	sCSVLine		: T_MaxString := '';(* Single CSV text line (row, record), we are using string as record buffer (your are able to see created fields) *)
	sCSVField		: T_MaxString := '';(* Single CSV field value (column, record field) *)
	//sCSVField		: UDINT;

	nRow	 		: UDINT 	:= 0;(* Row number (record) *)
	nColumn			: UDINT 	:= 0;(* Column number (record field) *)
	hFile			: UINT		:= 0;(* File handle of the source file *)
	step			: DWORD 	:= 0;
	fbFileOpen		: FB_FileOpen;(* Opens file *)
	fbFileClose		: FB_FileClose;(* Closes file *)
	fbFilePuts		: FB_FilePuts;(* Writes one record (line) *)
	fbFileWrite     : FB_FileWrite;
	fbWriter		: FB_CSVMemBufferWriter;(* Helper function block used to create CSV data bytes (single record line) *)
    StringModelWrite		: StringModel_256000_EX;
	fbFileRename			: FB_FileRename;//修改文件名称
	fbFileDelete			: FB_FileDelete;//删除文件
	writeTON				: TON;//延时写入

	(* :=[ (* Source PLC database *)
	'0_0', '0_1', '0_2', '0_3', '0_4', '0_5',
	'1_0', '1_1', '1_2', '1_3', '1_4', '1_5',
	'2_0', '2_1', '2_2', '2_3', '2_4', '2_5',
	'3_0', '3_1', '3_2', '3_3', '3_4', '3_5',
	'4_0', '4_1', '4_2', '4_3', '4_4', '4_5',
	'5_0', '5_1', '5_2', '5_3', '5_4', '5_5'];*)

END_VAR

DEFAULT_CSV_FIELD_SEP:= 16#2C;  //配置CSV文件的分割符，16#2C表明各个参数之间是用逗号分隔的。
CASE step OF
	0:(* Wait for rising edge at bWrite variable *)
		IF bWrite THEN
			bWrite 	:= FALSE;
			bBusy 	:= TRUE;
			error	:= FALSE;
			bError	:= FALSE;
			nErrId	:= 0;
			hFile	:= 0;
			nRow	:= 0;
			nColumn	:= 0;
			step 	:= 1;
		END_IF
	1:
		StringModelWrite.init();
		fbFileDelete(bExecute:= FALSE);
		fbFileRename(bExecute:= FALSE);
		step:=2;
	2:
		fbFileDelete(
			sNetId:= , 
			sPathName:= sFileNameOld, 
			ePath:= PATH_GENERIC, 
			bExecute:= TRUE, 
			tTimeout:= DEFAULT_ADS_TIMEOUT, 
			bBusy=> , 
			bError=> , 
			nErrId=> );
		step:=3;
	3:
		fbFileDelete(bExecute:= FALSE);
		IF NOT fbFileDelete.bBusy THEN
			step:=4;
		END_IF
	4:
		fbFileRename(
			sNetId:= , 
			sOldName:= sFileName, 
			sNewName:= sFileNameOld, 
			ePath:= PATH_GENERIC, 
			bExecute:= TRUE, 
			tTimeout:= DEFAULT_ADS_TIMEOUT, 
			bBusy=> , 
			bError=> , 
			nErrId=> );
		step:=5;
	5:
		fbFileRename(bExecute:= FALSE);
		IF NOT fbFileRename.bBusy THEN
			step:=10;
		END_IF

	10:(* Open source file *)
		fbFileOpen(  bExecute := FALSE  );
		fbFileOpen( sNetId := sNetId, sPathName := sFileName, nMode := FOPEN_MODEWRITE OR FOPEN_MODETEXT,(* Open file in TEXT mode! *)
					ePath := PATH_GENERIC, bExecute := TRUE );
		step := 20;

	20:(* Wait until open not busy *)
		//StringModelWrite.init();
		fbFileOpen( bExecute := FALSE, bError => bError, nErrID => nErrID, hFile => hFile );
		IF NOT fbFileOpen.bBusy THEN
			IF NOT fbFileOpen.bError THEN
				step := 30;
			ELSE(* Error: file not found? *)
				step := 1000;
			END_IF
		END_IF
	
	30:(* Convert one PLC record to CSV format *)
		FOR nRow:=0 TO csv_rows BY 1 DO
				sCSVLine := '';
				fbWriter.eCmd := eEnumCmd_First;(* Write first field value *)
			FOR nColumn := 0 TO csv_columns BY 1 DO
				sCSVField := STRING_TO_CSVFIELD( database[ nRow, nColumn ], FALSE );(* TODO: Get field value from your application *)
				(* Add new field to the record buffer *)
				fbWriter( 	pBuffer := ADR( sCSVLine ), cbBuffer := SIZEOF( sCSVLine ) - 1, putValue := sCSVField, pValue := 0, cbValue := 0,
							bCRLF := ( nColumn = csv_columns ) );(* bCRLF == TRUE => Write CRLF after the last field value *)
				IF fbWriter.bOk THEN
					fbWriter.eCmd := eEnumCmd_Next;(* Write next field value *)
				ELSE(* Error *)
					step := 1000;
					RETURN;
				END_IF
			END_FOR
			(* FB_FilePuts adds allready CR (carriage return) to the written line.
			We have to replace the $R$L characters with $L character to avoid double CR. *)
			IF RIGHT( sCSVLine, 2 ) = '$R$L' THEN
				sCSVLine := REPLACE( sCSVLine, '$L', 2, LEN( sCSVLine ) - 1 );
			END_IF
            StringModelWrite.append(str:= sCSVLine);
		END_FOR
		IF nRow> csv_rows THEN
			step := 40;(* Write record to the file *)
		END_IF
		writeTON(IN:=FALSE);

	40:(* Write record to file *)
		fbFileWrite( bExecute := FALSE );
		writeTON(IN:=NOT writeTON.Q,PT:=T#50MS);
		IF writeTON.Q THEN
			//fbFileWrite( sNetId := sNetId, hFile := hFile, pWriteBuff := StringModelWrite.getAddr, cbWriteLen := StringModelWrite.length, bExecute := TRUE );
			fbFileWrite( sNetId := sNetId, hFile := hFile, pWriteBuff := ADR(StringModelWrite.b), cbWriteLen := StringModelWrite.length, bExecute := TRUE );
			step := 50;
		END_IF

	50:(* Wait until write not busy *)
		fbFileWrite( bExecute := FALSE, bError => bError, nErrID => nErrID );
		IF NOT fbFileWrite.bBusy THEN
			IF NOT fbFileWrite.bError THEN
				step := 100;(* Write next record *)
			ELSE(* Error *)
				step := 1000;
			END_IF
		END_IF
		
	100:(* Close source file *)
		fbFileClose( bExecute := FALSE );
		fbFileClose( sNetId := sNetId, hFile := hFile, bExecute := TRUE );
		step := 110;

	110:(* Wait until close not busy *)
		fbFileClose( bExecute := FALSE, bError => bError, nErrID => nErrID );
		IF NOT fbFileClose.bBusy THEN
			hFile := 0;
			step := 1000;
		END_IF

	1000:(* Error or ready step => cleanup *)
		IF ( hFile <> 0 ) THEN
			step := 100; (* Close the source file *)
		ELSE
			bBusy := FALSE;
			error := bError;
			step := 0;	(* Ready *)
		END_IF
END_CASE

END_FUNCTION_BLOCK

// ---- POUs/BaseModule/DataSaveModule_EX/csvReadWriteInTextMode/StringModel_256000_EX.TcPOU
FUNCTION_BLOCK StringModel_256000_EX
VAR CONSTANT
	cNumLength:UDINT:=gMaxNumLength;//maximum -+21 4748 3647
	cNumBegin:UDINT:=gNumBegin;
END_VAR
VAR_INPUT
END_VAR
VAR_OUTPUT
	length:UDINT;
	error:BOOL;
	b:ARRAY[cNumBegin..(cNumLength+cNumBegin-1)]OF BYTE;
END_VAR
VAR
	//b:ARRAY[cNumBegin..(cNumLength+cNumBegin-1)]OF BYTE;	
	endPoint:UDINT:=cNumBegin;
END_VAR

(*
	version 1.0 hjm in Zhuhai IA 20171122

	to save string to byte array
*)

METHOD append 
VAR_INPUT
	str:STRING(255);
END_VAR
VAR
	i:INT;
	strTemp:STRING(1);
	_leng:INT;
END_VAR

_leng:=LEN(str);
FOR i:=1 TO _leng DO
	strTemp:=LEFT(str,1);
	str:= DELETE (str,1,1);
	IF endPoint<=cNumLength THEN
		b[endPoint]:=F_ToASC(strTemp);
		endPoint:=endPoint+1;	
	ELSE
		error:=TRUE;
		RETURN;	
	END_IF
END_FOR
length:=endPoint-cNumBegin;
END_METHOD

METHOD getAddr:POINTER TO BYTE;
getAddr:=ADR(b);
END_METHOD

METHOD init 
VAR_INPUT
END_VAR
VAR
	i:UDINT;
END_VAR
FOR i:=cNumBegin TO (cNumLength+cNumBegin-1) DO
	b[i]:=0;
END_FOR
endPoint:=cNumBegin;
error:=FALSE;
END_METHOD

METHOD reset 
VAR_INPUT
END_VAR
endPoint:=cNumBegin;
error:=FALSE;
END_METHOD

END_FUNCTION_BLOCK

// ---- POUs/BaseModule/DataSaveModule_EX/csvReadWriteInTextMode/P_TextModeRead.TcPOU
FUNCTION_BLOCK P_TextModeRead
VAR_IN_OUT
	database		: ARRAY[0..gMAX_CSV_ROWS, 0..gMAX_CSV_COLUMNS ] OF STRING(30);(* Target PLC database *)
	csv_rows		: UDINT;
	csv_columns		: UDINT;
END_VAR
VAR_INPUT
	bRead			: BOOL := FALSE;(* Rising edge starts program execution *)	
	sFileName		: T_MaxString := '';(* CSV source file path and name *)
END_VAR
VAR_OUTPUT
	bBusy			: BOOL;
	error			: BOOL;
	nErrId			: UDINT;	
END_VAR
VAR
	bError			: BOOL;
	sNetId			: T_AmsNetId := '';	(* TwinCAT system network address *)
	sCSVLine		: T_MaxString := '';(* Single CSV text line (row, record), we are using string as record buffer (your are able to see read fields)  *)
	sCSVField		: T_MaxString := '';(* Single CSV field value (column, record field) *)
	nRow	 		: UDINT 	:= 0;(* Row number (record) *)
	nColumn			: UDINT 	:= 0;(* Column number (record field) *)
	hFile			: UINT		:= 0;(* File handle of the source file *)
	step			: DWORD 	:= 0;
	fbFileOpen		: FB_FileOpen;(* Opens file *)
	fbFileClose		: FB_FileClose;(* Closes file *)
	fbFileGets		: FB_FileGets;(* Reads one record (line) *)
	fbFileRead		: FB_FileRead;//---------------------------------------
	fbReader		: FB_CSVMemBufferReader;(* Helper function block used to parse CSV data bytes (single record line) *)
	
	readData:ARRAY[gNumBegin..(gMaxNumLength+gNumBegin-1)]OF BYTE;
	strTemp : T_MaxString;
	strT : T_MaxString;
	i : UDINT:=0;
	iTemp : UDINT:=0;
END_VAR

DEFAULT_CSV_FIELD_SEP:= 16#2C;  //配置CSV文件的分割符，16#2C表明各个参数之间是用逗号分隔的。
CASE step OF
	0:	(* Wait for rising edge at bRead variable *)
		IF bRead THEN
			bRead 	:= FALSE;
			bBusy 	:= TRUE;
			error:= bError	:= FALSE;
			nErrId	:= 0;
			hFile	:= 0;
			nRow	:= 0;
			nColumn	:= 0;
			MEMSET( ADR( database ), 0, SIZEOF( database ) );
			step 		:= 1;
		END_IF

	1:	(* Open source file *)
		fbFileOpen(  bExecute := FALSE  );
		fbFileOpen( sNetId := sNetId, sPathName := sFileName, nMode := FOPEN_MODEREAD OR FOPEN_MODETEXT,(* Open file in TEXT mode! *)
					ePath := PATH_GENERIC, bExecute := TRUE );
		step := 2;

	2:(* Wait until open not busy *)
		fbFileOpen( bExecute := FALSE, bError => bError, nErrID => nErrID, hFile => hFile );
		IF NOT fbFileOpen.bBusy THEN
			IF NOT fbFileOpen.bError THEN
				step := 3;
			ELSE(* Error: file not found? *)
				step := 100;
			END_IF
		END_IF
		
	3:
		step := 4;
	4:
		fbFileRead(
			sNetId:= sNetId, 
			hFile:= hFile, 
			bExecute:= FALSE,);
		step := 5;
	5:(*Read data from file*)
		fbFileRead(
			sNetId:= sNetId, 
			hFile:= hFile, 
			pReadBuff:= ADR(readData),
			cbReadLen:= gMaxNumLength,
			bExecute:= TRUE, 
			tTimeout:= , 
			bBusy=> , 
			bError=> , 
			nErrId=> , 
			cbRead=> , 
			bEOF=> );
		IF NOT fbFileRead.bBusy AND NOT fbFileRead.bError THEN
			IF fbFileRead.bEOF THEN
				step := 6;
			END_IF
			step := 6;
			fbFileRead(
				sNetId:= sNetId, 
				hFile:= hFile, 
				bExecute:= FALSE,);
		ELSIF fbFileRead.bError THEN
			step := 100;
		END_IF
		sCSVLine := '';
		iTemp:=1;
	6:
		FOR nRow:=0 TO csv_rows BY 1 DO
			sCSVLine := '';
			FOR i:=iTemp TO gMaxNumLength BY 1 DO
				strT := F_ToCHR(c:=readData[i]);
				IF '$L' = strT THEN
					strTemp:=CONCAT(STR1:=sCSVLine,STR2:='$R$L');
					iTemp:=i+1;
					EXIT;
				ELSE
					sCSVLine:=CONCAT(STR1:=sCSVLine,STR2:=strT);
				END_IF
			END_FOR
			fbReader.eCmd := eEnumCmd_First;(* Read first field value *)
			FOR nColumn := 0 TO csv_columns BY 1 DO
				fbReader( pBuffer := ADR( sCSVLine ), cbBuffer := SIZEOF( sCSVLine ), getValue => sCSVField);
				IF fbReader.bOk THEN
					fbReader.eCmd := eEnumCmd_Next;
					IF ( nRow <= csv_rows ) THEN
						IF ( nColumn <= csv_columns ) THEN
							database[nRow, nColumn] := CSVFIELD_TO_STRING( sCSVField, FALSE );
						END_IF
					END_IF
				END_IF
			END_FOR
			IF fbReader.bCRLF THEN(* CRLF == TRUE => End of reacord reached *)
				nColumn := 0;
			END_IF
		END_FOR
		step := 10;

	10:	(* Close source file *)
		fbFileClose( bExecute := FALSE );
		fbFileClose( sNetId := sNetId, hFile := hFile, bExecute := TRUE );
		step := 11;

	11:(* Wait until close not busy *)
		fbFileClose( bExecute := FALSE, bError => bError, nErrID => nErrID );
		IF ( NOT fbFileClose.bBusy ) THEN
			hFile := 0;
			step := 100;
		END_IF

	100: (* Error or ready step => cleanup *)
		IF ( hFile <> 0 ) THEN
			step := 10; (* Close the source file *)
		ELSE
			bBusy := FALSE;
			error := bError;
			step := 0;	(* Ready *)
		END_IF

END_CASE

END_FUNCTION_BLOCK

// ---- POUs/BaseModule/DataSaveModule_EX/RecipeSaveModule_EX.TcPOU
FUNCTION_BLOCK RecipeSaveModule_EX
VAR_INPUT
	sFileName						:T_MaxString:='C:\IASaveData.csv';//'Hard Disk\IASaveData.csv'  数据文件存储路径
	readB							:BOOL:=FALSE;//读取触发
	saveB							:BOOL:=FALSE;//保存触发
	saveAct							:BOOL:=FALSE;//保存触发
	deleteB							:BOOL:=FALSE;// 删除触发
	recipeStepDelete				:BOOL:=FALSE;// 删除触发
	dataString						:ARRAY[0..gRecipeMAX_CSV_ROWS, 0..gRecipeMAX_CSV_COLUMNS ] OF STRING(30);//BOOL数据源
	pDatabaseHMI					:ARRAY[1..gRecipeMAX_CSV_ROWS+1] OF RecipePar;(* Target PLC database *)
	pDatabase						:ARRAY[0..gRecipeMAX_CSV_ROWS, 0..gRecipeMAX_CSV_COLUMNS ] OF STRING(30);(* Target PLC database *)
	dataStringLength				:UDINT:=gRecipeMAX_CSV_ROWS;
	dataStringLengthRead			:UDINT:=gRecipeMAX_CSV_ROWS;
END_VAR
VAR_OUTPUT
	busy							:BOOL:=FALSE;
	rDone							:BOOL:=FALSE;
	sDone							:BOOL:=FALSE;
	error							:BOOL:=FALSE;
	errID							:UDINT:=0;
	errTxt							:STRING(255):='';
	outData							:ARRAY [1..gRecipeMAX_String_NUM] OF RecipePar; 
	checkFileExistError				:BOOL;
END_VAR
VAR_IN_OUT
	
END_VAR
VAR	
	saveActStep						:INT;//保存触发步数
	csv_rows						:UDINT:=gRecipeMAX_CSV_ROWS;
	csv_columns						:UDINT:=gRecipeMAX_CSV_COLUMNS;
	startUpB						:BOOL:=FALSE;
	writeTxt						:P_TextModeWrite_Recipe;
	readTxt							:P_TextModeRead_Recipe;
	deleteTxt						:P_TextModeDelete_1;
	fbFileOpen						:FB_FileOpen;//检查文件是否存在
	fbFileClose						:FB_FileClose;(* Closes file *)
	hFile							:UINT:=0;(* File handle of the source file *)
	initB							:BOOL:=FALSE;
	saveStep						:UINT:=0;
	deleteStep						:UINT:=0;
	readStep						:UINT:=0;
	sFileNameOld					:T_MaxString;//旧文件名
//获取系统时间
	ntGetTime				: NT_GetTime;
	systemTimeStruct		: TIMESTRUCT;
	getSystemTimeStep		: UINT:=0;
	systemTIMEStr			: STRING:='';//系统时间，格式YYYY-MM-DD hh:mm:ss_zzz
	systemTIMEStr2			: STRING:='';//系统时间，格式YYYYMMDDhhmmss
	sysTIMEStrYY			: STRING:='';//系统时间，年
	sysTIMEStrMM			: STRING:='';//系统时间，月
	sysTIMEStrDD			: STRING:='';//系统时间，日
	sysTIMEStr_HH			: STRING:='';//系统时间，时
	sysTIMEStr_mm			: STRING:='';//系统时间，分
	sysTIMEStr_ss			: STRING:='';//系统时间，秒
	itemp:INT;
	ton1:TON;
	remainber:INT;
END_VAR


csv_rows:=dataStringLength + 1;
IF dataStringLength>gRecipeMAX_String_NUM THEN
	dataStringLength:=gRecipeMAX_String_NUM;
END_IF
IF csv_rows>gRecipeMAX_CSV_ROWS THEN
	csv_rows:=gRecipeMAX_CSV_ROWS;
END_IF

//judge length
IF gRecipeMAX_CSV_ROWS<(dataStringLength+1) THEN
	error:=TRUE;
	errTxt:='dataBase$'s length too short';
	RETURN;
END_IF
IF csv_rows<(dataStringLength+1) THEN
	error:=TRUE;
	errTxt:='dataBase$'s length too short';
	RETURN;
END_IF

init();
IF initB THEN
	saveActRun();
	readMethod();
	saveMethod();
	deleteMethod();
	DeleteRecipeStep();
END_IF
getSystemTime();

METHOD addRecipeStep : BOOL
VAR_INPUT
	index:INT;
END_VAR
pDatabase[index,0]:=INT_TO_STRING(gShowNum);//num
pDatabase[index,1]:='1';//data type
pDatabase[index,2]:=gRecipeShowNameNow;;//name
pDatabase[index,3]:=INT_TO_STRING(gShowNum);// Step
pDatabase[index,4]:='0';//par1
pDatabase[index,5]:='0';//par2
pDatabase[index,6]:='0';//par3
pDatabase[index,7]:='0';//par4
pDatabase[index,8]:='0';//par5
pDatabase[index,9]:='0';//par6
pDatabase[index,10]:='0';//par7
pDatabase[index,11]:='0';//par8
pDatabase[index,12]:='0';//par9
pDatabase[index,13]:='0';//par10
pDatabase[index,14]:='0';//par11
pDatabase[index,15]:='0';//par12
pDatabase[index,16]:='0';//par13
pDatabase[index,17]:='0';//par14
pDatabase[index,18]:='0';//par15

gRecipeViewData[index].NUM:=INT_TO_STRING(gShowNum);
gRecipeViewData[index].etchTime:='0';
gRecipeViewData[index].rfPoint_Source:='0';
gRecipeViewData[index].pdvPoint:='0';
gRecipeViewData[index].mfc1:='0';
gRecipeViewData[index].mfc2:='0';
gRecipeViewData[index].mfc3:='0';
gRecipeViewData[index].mfc4:='0';
gRecipeViewData[index].mfc5:='0';
gRecipeViewData[index].mfc6:='0';
gRecipeViewData[index].mfc7:='0';
gRecipeViewData[index].mfc8:='0';
gRecipeViewData[index].mfc9:='0';
gRecipeViewData[index].rfPoint_Power:='0';
gRecipeViewData[index].par_2:='0';
gRecipeViewData[index].par_3:='0';

gRecipeEditorData[index].NUM:=INT_TO_STRING(gShowNum);
gRecipeEditorData[index].etchTime:='0';
gRecipeEditorData[index].rfPoint_Source:='0';
gRecipeEditorData[index].pdvPoint:='0';
gRecipeEditorData[index].mfc1:='0';
gRecipeEditorData[index].mfc2:='0';
gRecipeEditorData[index].mfc3:='0';
gRecipeEditorData[index].mfc4:='0';
gRecipeEditorData[index].mfc5:='0';
gRecipeEditorData[index].mfc6:='0';
gRecipeEditorData[index].mfc7:='0';
gRecipeEditorData[index].mfc8:='0';
gRecipeEditorData[index].mfc9:='0';
gRecipeEditorData[index].rfPoint_Power:='0';
gRecipeEditorData[index].par_2:='0';
gRecipeEditorData[index].par_3:='0';
END_METHOD

METHOD addSlector : BOOL

VAR_INPUT
	newName							:STRING;
END_VAR
VAR_OUTPUT
	error:BOOL;
END_VAR
VAR_IN_OUT
	outrecipeSelect					:ARRAY [1..gRecipeNameMAX_String_NUM+1] OF RecipeShowStr;
	outrecipeSelectShow				:ARRAY [1..10] OF RecipeShowStr;
END_VAR
VAR
	itemp:INT;
END_VAR
IF (len(newName)>0) THEN
	FOR itemp:=UDINT_TO_INT(gRecipeNameMAX_String_NUM)+1 TO gRecipeSelctMaxIndex+2 BY 1 DO
		outrecipeSelect[itemp].Name:=outrecipeSelect[itemp-1].Name;
	END_FOR
	outrecipeSelect[gRecipeSelctMaxIndex+1].Name:=newName;
	
	FOR itemp:=UDINT_TO_INT(gRecipeNameMAX_String_NUM)+1 TO gRecipeSelctMaxIndex+1 BY 1 DO
		outrecipeSelectShow[itemp].Name:=outrecipeSelectShow[itemp-1].Name;
	END_FOR
	outrecipeSelectShow[gRecipeSelctMaxIndex].Name:=newName;
	
	gRecipeSelctMaxIndex:=gRecipeSelctMaxIndex+1;
	
	gRecipeSelectIndex1:=gRecipeSelctMaxIndex;
	
	error:=FALSE;
ELSE
	error:=TRUE;
END_IF
END_METHOD

METHOD PRIVATE createDir : BOOL
VAR
	sPathNameTemp	: T_MaxString := 'C:\TwinCAT\Data.txt';
	sDriveTemp		: STRING(3);
	sDirTemp		: T_MaxString;
	sFileNameTemp	: T_MaxString;
	sExtTemp		: T_MaxString;
	bSuccess		: BOOL;
	fbCreateDir		: FB_CreateDir;
	fbCreateDir2	: FB_CreateDir;
	sFileDirTemp	: T_MaxString;
	sFileDirTemp2	: T_MaxString;
END_VAR
sPathNameTemp:=sFileName;
bSuccess := F_SplitPathName( sPathName := sPathNameTemp,
	sDrive := sDriveTemp,
	sDir := sDirTemp,
	sFileName := sFileNameTemp,
	sExt := sExtTemp );
IF bSuccess THEN
	bSuccess:=FALSE;
	IF LEFT(sDirTemp,LEN(sDirTemp)-1) <> '' THEN
		//sFileDirTemp:=CONCAT(STR1:=sDriveTemp,STR2:=LEFT(sDirTemp,LEN(sDirTemp)-1));
		//sFileNameOld:=CONCAT(STR1:=sFileDirTemp,STR2:=CONCAT('\',CONCAT(sFileNameTemp,'_Old.csv')));//用于重命名参数文件
		sFileDirTemp:='';
		sFileDirTemp:=CONCAT(sFileDirTemp,sDriveTemp);
		sFileDirTemp:=CONCAT(sFileDirTemp,LEFT(sDirTemp,LEN(sDirTemp)-1));
		sFileDirTemp2:='';
		sFileDirTemp2:=CONCAT(sFileDirTemp2,sFileDirTemp);
		sFileDirTemp2:=CONCAT(sFileDirTemp2,'\Old');
		
		sFileNameOld:='';
		sFileNameOld:=CONCAT(sFileNameOld,sFileDirTemp);
		sFileNameOld:=CONCAT(sFileNameOld,'\Old\');//'\'
		sFileNameOld:=CONCAT(sFileNameOld,sFileNameTemp);
		sFileNameOld:=CONCAT(sFileNameOld,'_Old_');
		sFileNameOld:=CONCAT(sFileNameOld,systemTIMEStr2);
		sFileNameOld:=CONCAT(sFileNameOld,'.csv');
		
		fbCreateDir(
			sNetId:= , 
			sPathName:= sFileDirTemp, 
			ePath:= PATH_GENERIC, 
			bExecute:= TRUE, 
			tTimeout:= , 
			bBusy=> , 
			bError=> , 
			nErrId=> );
		fbCreateDir2(
			sNetId:= , 
			sPathName:= sFileDirTemp2, 
			ePath:= PATH_GENERIC, 
			bExecute:= TRUE, 
			tTimeout:= , 
			bBusy=> , 
			bError=> , 
			nErrId=> );
	END_IF
END_IF
fbCreateDir(
	sNetId:= , 
	sPathName:= , 
	ePath:= , 
	bExecute:= FALSE, 
	tTimeout:= , 
	bBusy=> , 
	bError=> , 
	nErrId=> );
fbCreateDir2(
	sNetId:= , 
	sPathName:= , 
	ePath:= , 
	bExecute:= FALSE, 
	tTimeout:= , 
	bBusy=> , 
	bError=> , 
	nErrId=> );
END_METHOD

METHOD PRIVATE data2String : BOOL
VAR_INPUT
END_VAR
VAR
	i:UDINT:=0;
END_VAR
//judge length
IF gRecipeMAX_CSV_ROWS<(gRecipeMAX_String_NUM+1) THEN
	error:=TRUE;
	errTxt:='dataBase$'s length too short';
	RETURN;
END_IF
IF csv_rows<(dataStringLength+1) THEN
	error:=TRUE;
	errTxt:='dataBase$'s length too short';
	RETURN;
END_IF

//bool
FOR i:=0 TO gShowNum DO
	//////////1
	pDatabase[i+1,2]:=gRecipeShowNameNow;
	IF LEN(gRecipeEditorData[i+1].etchTime)>0 THEN
		IF IsAllDigits(gRecipeEditorData[i+1].etchTime) THEN
			pDatabase[i+1,4]:=gRecipeEditorData[i+1].etchTime;//Par1
		ELSE
			error_Trigger(10);
		END_IF
	ELSE
		pDatabase[i+1,4]:='0';
	END_IF
	///////////////2
	IF LEN(gRecipeEditorData[i+1].rfPoint_Source)>0 THEN
		IF IsAllDigits(gRecipeEditorData[i+1].rfPoint_Source) THEN
			pDatabase[i+1,5]:=gRecipeEditorData[i+1].rfPoint_Source;//Par2
		ELSE
			error_Trigger(11);
		END_IF
	ELSE
		pDatabase[i+1,5]:='0';
	END_IF
	///////////////////////3
	
	IF LEN(gRecipeEditorData[i+1].pdvPoint)>0 THEN
		IF IsAllDigits(gRecipeEditorData[i+1].pdvPoint) THEN
			pDatabase[i+1,6]:=gRecipeEditorData[i+1].pdvPoint;//Par3
		ELSE
			error_Trigger(12);
		END_IF
	ELSE
		pDatabase[i+1,6]:='0';
	END_IF
	/////////////////
	
	IF LEN(gRecipeEditorData[i+1].mfc1)>0 THEN
		IF IsAllDigits(gRecipeEditorData[i+1].mfc1) THEN
			pDatabase[i+1,7]:=gRecipeEditorData[i+1].mfc1;//Par4
		ELSE
			error_Trigger(13);
		END_IF
		
	ELSE
		pDatabase[i+1,7]:='0';
	END_IF
	//////////////////
	
	IF LEN(gRecipeEditorData[i+1].mfc2)>0 THEN
		IF IsAllDigits(gRecipeEditorData[i+1].mfc2) THEN
			pDatabase[i+1,8]:=gRecipeEditorData[i+1].mfc2;//Par5
		ELSE
			error_Trigger(14);
		END_IF
		
	ELSE
		pDatabase[i+1,8]:='0';
	END_IF
	/////////////////
	
	IF LEN(gRecipeEditorData[i+1].mfc3)>0 THEN
		IF IsAllDigits(gRecipeEditorData[i+1].mfc3) THEN
			pDatabase[i+1,9]:=gRecipeEditorData[i+1].mfc3;//Par6
		ELSE
			error_Trigger(15);
		END_IF
		
	ELSE
		pDatabase[i+1,9]:='0';
	END_IF
	////////////////
	
	IF LEN(gRecipeEditorData[i+1].mfc4)>0 THEN
		IF IsAllDigits(gRecipeEditorData[i+1].mfc4) THEN
			pDatabase[i+1,10]:=gRecipeEditorData[i+1].mfc4;//Par7
		ELSE
			error_Trigger(16);
		END_IF
		
	ELSE
		pDatabase[i+1,10]:='0';
	END_IF
	//////////////////////
	
	IF LEN(gRecipeEditorData[i+1].mfc5)>0 THEN
		IF IsAllDigits(gRecipeEditorData[i+1].mfc5) THEN
			pDatabase[i+1,11]:=gRecipeEditorData[i+1].mfc5;//Par8
		ELSE
			error_Trigger(17);
		END_IF
		
	ELSE
		pDatabase[i+1,11]:='0';
	END_IF
	//////////////////
	
	IF LEN(gRecipeEditorData[i+1].mfc6)>0 THEN
		IF IsAllDigits(gRecipeEditorData[i+1].mfc6) THEN
			pDatabase[i+1,12]:=gRecipeEditorData[i+1].mfc6;//Par9
		ELSE
			error_Trigger(18);
		END_IF
		
	ELSE
		pDatabase[i+1,12]:='0';
	END_IF
	///////////////////
	
	IF LEN(gRecipeEditorData[i+1].mfc7)>0 THEN
		IF IsAllDigits(gRecipeEditorData[i+1].mfc7) THEN
			pDatabase[i+1,13]:=gRecipeEditorData[i+1].mfc7;//Par10
		ELSE
			error_Trigger(19);
		END_IF
		
	ELSE
		pDatabase[i+1,13]:='0';
	END_IF
	//////////////////
	
	IF LEN(gRecipeEditorData[i+1].mfc8)>0 THEN
		IF IsAllDigits(gRecipeEditorData[i+1].mfc8) THEN
			pDatabase[i+1,14]:=gRecipeEditorData[i+1].mfc8;//Par11
		ELSE
			error_Trigger(20);
		END_IF
		
	ELSE
		pDatabase[i+1,14]:='0';
	END_IF
	///////////////////
	
	IF LEN(gRecipeEditorData[i+1].mfc9)>0 THEN
		IF IsAllDigits(gRecipeEditorData[i+1].mfc9) THEN
			pDatabase[i+1,15]:=gRecipeEditorData[i+1].mfc9;//Par12
		ELSE
			error_Trigger(21);
		END_IF
		
	ELSE
		pDatabase[i+1,15]:='0';
	END_IF
	////////////////////
	
	IF LEN(gRecipeEditorData[i+1].rfPoint_Power)>0 THEN
		IF IsAllDigits(gRecipeEditorData[i+1].rfPoint_Power) THEN
			pDatabase[i+1,16]:=gRecipeEditorData[i+1].rfPoint_Power;//Par13
		ELSE
			error_Trigger(22);
		END_IF
		
	ELSE
		pDatabase[i+1,16]:='0';
	END_IF
	/////////////////////
	
	IF LEN(gRecipeEditorData[i+1].par_2)>0 THEN
		IF IsAllDigits(gRecipeEditorData[i+1].par_2) THEN
			pDatabase[i+1,17]:=gRecipeEditorData[i+1].par_2;//Par14
		ELSE
			error_Trigger(23);
		END_IF
		
	ELSE
		pDatabase[i+1,17]:='0';
	END_IF
	////////////////////
	
	IF LEN(gRecipeEditorData[i+1].par_3)>0 THEN
		IF IsAllDigits(gRecipeEditorData[i+1].par_3) THEN
			pDatabase[i+1,18]:=gRecipeEditorData[i+1].par_3;//Par15
		ELSE
			error_Trigger(24);
		END_IF
		
	ELSE
		pDatabase[i+1,18]:='0';
	END_IF
	
END_FOR
END_METHOD

METHOD PRIVATE deleteMethod : BOOL
VAR_INPUT
END_VAR
CASE deleteStep OF
0:
	IF deleteB AND (NOT busy) THEN
		deleteStep:=1;
		deleteB:=FALSE;
		busy:=TRUE;
		sDone:=FALSE;
		error:=FALSE;
		errID:=0;
		errTxt:='';
	END_IF

1:
	deleteStep:=2;

2:
	deleteTxt(
	bDelete:=TRUE , 
	sFileName:=sFileName , 
	sFileNameOld:= , 
	bBusy=> , 
	error=> , 
	nErrId=> );	
	deleteStep:=3;

3:
	deleteTxt.bDelete:=FALSE;
	
	IF error THEN
		deleteStep:=110;
		RETURN;
	END_IF

	IF NOT writeTxt.bBusy THEN
		deleteStep:=100;
	END_IF

100:
	busy:=FALSE;
	sDone:=TRUE;
	error:=error;
	errID:=errID;
	errTxt:=errTxt;

	IF NOT deleteB THEN
		deleteStep:=0;
	END_IF

110:
	busy:=FALSE;
	sDone:=FALSE;
	error:=TRUE;
	errID:=errID;
	errTxt:='save data fail';

	IF NOT deleteB THEN
		deleteStep:=0;
	END_IF
END_CASE
deleteTxt(
	bDelete:= , 
	sFileName:=sFileName , 
	sFileNameOld:= , 
	bBusy=> , 
	error=> , 
	nErrId=> );
END_METHOD

ACTION DeleteRecipeStep:
IF recipeStepDelete THEN
	IF gselectRow>0 AND gselectRow<=UDINT_TO_INT(gRecipeMAX_String_NUM) THEN
		FOR itemp:=gselectRow TO UDINT_TO_INT(gRecipeMAX_String_NUM-1) BY 1 DO
			gRecipeEditorData[itemp].NUM:=gRecipeEditorData[itemp+1].NUM;
			gRecipeEditorData[itemp].etchTime:=gRecipeEditorData[itemp+1].etchTime;
			gRecipeEditorData[itemp].rfPoint_Source:=gRecipeEditorData[itemp+1].rfPoint_Source;
			gRecipeEditorData[itemp].pdvPoint:=gRecipeEditorData[itemp+1].pdvPoint;
			gRecipeEditorData[itemp].mfc1:=gRecipeEditorData[itemp+1].mfc1;
			gRecipeEditorData[itemp].mfc2:=gRecipeEditorData[itemp+1].mfc2;
			gRecipeEditorData[itemp].mfc3:=gRecipeEditorData[itemp+1].mfc3;
			gRecipeEditorData[itemp].mfc4:=gRecipeEditorData[itemp+1].mfc4;
			gRecipeEditorData[itemp].mfc5:=gRecipeEditorData[itemp+1].mfc5;
			gRecipeEditorData[itemp].mfc6:=gRecipeEditorData[itemp+1].mfc6;
			gRecipeEditorData[itemp].mfc7:=gRecipeEditorData[itemp+1].mfc7;
			gRecipeEditorData[itemp].mfc8:=gRecipeEditorData[itemp+1].mfc8;
			gRecipeEditorData[itemp].mfc9:=gRecipeEditorData[itemp+1].mfc9;
			gRecipeEditorData[itemp].rfPoint_Power:=gRecipeEditorData[itemp+1].rfPoint_Power;
			gRecipeEditorData[itemp].par_2:=gRecipeEditorData[itemp+1].par_2;
			gRecipeEditorData[itemp].par_3:=gRecipeEditorData[itemp+1].par_3;
			gRecipeEditorData[itemp].par_4:=gRecipeEditorData[itemp+1].par_4;
		END_FOR
		gRecipeEditorData[gShowNum].NUM:='';
		gRecipeEditorData[gShowNum].etchTime:='';
		gRecipeEditorData[gShowNum].rfPoint_Source:='';
		gRecipeEditorData[gShowNum].pdvPoint:='';
		gRecipeEditorData[gShowNum].mfc1:='';
		gRecipeEditorData[gShowNum].mfc2:='';
		gRecipeEditorData[gShowNum].mfc3:='';
		gRecipeEditorData[gShowNum].mfc4:='';
		gRecipeEditorData[gShowNum].mfc5:='';
		gRecipeEditorData[gShowNum].mfc6:='';
		gRecipeEditorData[gShowNum].mfc7:='';
		gRecipeEditorData[gShowNum].mfc8:='';
		gRecipeEditorData[gShowNum].mfc9:='';
		gRecipeEditorData[gShowNum].rfPoint_Power:='';
		gRecipeEditorData[gShowNum].par_2:='';
		gRecipeEditorData[gShowNum].par_3:='';
		gRecipeEditorData[gShowNum].par_4:='';
		pDatabase[gShowNum,0]:='';
		pDatabase[gShowNum,1]:='';
		pDatabase[gShowNum,2]:='';
		pDatabase[gShowNum,3]:='';
		pDatabase[gShowNum,5]:='';
		pDatabase[gShowNum,6]:='';
		pDatabase[gShowNum,7]:='';
		pDatabase[gShowNum,8]:='';
		pDatabase[gShowNum,9]:='';
		pDatabase[gShowNum,10]:='';
		pDatabase[gShowNum,11]:='';
		pDatabase[gShowNum,12]:='';
		pDatabase[gShowNum,13]:='';
		pDatabase[gShowNum,14]:='';
		pDatabase[gShowNum,15]:='';
		pDatabase[gShowNum,16]:='';
		pDatabase[gShowNum,17]:='';
		pDatabase[gShowNum,18]:='';
		pDatabase[gShowNum,19]:='';

	gShowNum:=gShowNum-1;
	IF gShowNum<0 THEN
		gShowNum:=0;
		error_Trigger(30);
	END_IF
	gRecipeViewData:=gRecipeEditorData;
		
	END_IF
	recipeStepDelete:=FALSE;
END_IF
END_ACTION

METHOD deleteSlector : BOOL

VAR_INPUT
	recipeSelect					:ARRAY [1..gRecipeNameMAX_String_NUM+1] OF RecipeShowStr;
	recipeSelectShow				:ARRAY [1..10] OF RecipeShowStr;
	inidex							:INT;
END_VAR
VAR_OUTPUT
	error:BOOL;
	outrecipeSelect					:ARRAY [1..gRecipeNameMAX_String_NUM+1] OF RecipeShowStr;
	outrecipeSelectShow				:ARRAY [1..10] OF RecipeShowStr;
END_VAR
VAR
	itemp:INT;
END_VAR
outrecipeSelect:=recipeSelect;
outrecipeSelectShow:=recipeSelectShow;
IF inidex>0 AND inidex<=gRecipeSelctMaxIndex THEN
	FOR itemp:=inidex TO UDINT_TO_INT(gRecipeNameMAX_String_NUM) BY 1 DO
		outrecipeSelect[itemp].Name:=outrecipeSelect[itemp+1].Name;
	END_FOR
	outrecipeSelect[gRecipeNameMAX_String_NUM+1].Name:='';
	
	FOR itemp:=inidex TO gRecipeSelctMaxIndex-1 BY 1 DO
		outrecipeSelectShow[itemp].Name:=outrecipeSelectShow[itemp+1].Name;
	END_FOR
	outrecipeSelectShow[gRecipeSelctMaxIndex].Name:='';
	
	gRecipeSelctMaxIndex:=gRecipeSelctMaxIndex-1;
	
	gRecipeSelectIndex1:=1;
	
	error:=FALSE;
ELSE
	error:=TRUE;
END_IF
END_METHOD

METHOD PRIVATE getSystemTime : BOOL
VAR_INPUT
END_VAR
//获取本地系统时间--输出到变量 systemTIMEStr
CASE getSystemTimeStep OF
0:
	ntGetTime(
		NETID:= , 
		START:= FALSE, 
		TMOUT:= , 
		BUSY=> , 
		ERR=> , 
		ERRID=> , 
		TIMESTR=> systemTimeStruct);
	IF NOT ntGetTime.BUSY AND NOT ntGetTime.ERR THEN
		getSystemTimeStep:=getSystemTimeStep+1;
	END_IF
1:
	ntGetTime(
		NETID:= , 
		START:= TRUE, 
		TMOUT:= , 
		BUSY=> , 
		ERR=> , 
		ERRID=> , 
		TIMESTR=> systemTimeStruct);
	IF NOT ntGetTime.BUSY AND NOT ntGetTime.ERR THEN
		systemTIMEStr:=SYSTEMTIME_TO_STRING(systemTimeStruct);//系统时间转成字符串格式
		
		sysTIMEStrYY:=WORD_TO_DECSTR(in:=systemTimeStruct.wYear,iPrecision:=4);
		sysTIMEStrMM:=WORD_TO_DECSTR(in:=systemTimeStruct.wMonth,iPrecision:=2);
		sysTIMEStrDD:=WORD_TO_DECSTR(in:=systemTimeStruct.wDay,iPrecision:=2);
		sysTIMEStr_HH:=WORD_TO_DECSTR(in:=systemTimeStruct.wHour,iPrecision:=2);
		sysTIMEStr_mm:=WORD_TO_DECSTR(in:=systemTimeStruct.wMinute,iPrecision:=2);
		sysTIMEStr_ss:=WORD_TO_DECSTR(in:=systemTimeStruct.wSecond,iPrecision:=2);
		
		systemTIMEStr2:='';
		systemTIMEStr2:=CONCAT(systemTIMEStr2,sysTIMEStrYY);
		systemTIMEStr2:=CONCAT(systemTIMEStr2,sysTIMEStrMM);
		systemTIMEStr2:=CONCAT(systemTIMEStr2,sysTIMEStrDD);
		systemTIMEStr2:=CONCAT(systemTIMEStr2,sysTIMEStr_HH);
		systemTIMEStr2:=CONCAT(systemTIMEStr2,sysTIMEStr_mm);
		systemTIMEStr2:=CONCAT(systemTIMEStr2,sysTIMEStr_ss);
		
		getSystemTimeStep:=0;
	ELSIF ntGetTime.ERR THEN
		systemTIMEStr:='';
		getSystemTimeStep:=0;
	END_IF	
END_CASE
END_METHOD

METHOD getValue : BOOL
VAR_IN_OUT
	value:STRING;
END_VAR
VAR_INPUT
	cnum:UDINT;
	rnum:UDINT;
END_VAR
IF 0<=rnum AND rnum<=dataStringLength
	AND 0<=cnum AND cnum<=gRecipeMAX_CSV_COLUMNS THEN
	value:=pDatabase[rnum,cnum];
	getValue:=TRUE;
ELSE
	value:='';
	getValue:=FALSE;
END_IF
END_METHOD

METHOD PRIVATE init : BOOL
VAR_INPUT
END_VAR
VAR
	i:UDINT:=0;
END_VAR
//创建生成初始表格
//judge length
IF gRecipeMAX_CSV_ROWS<(gRecipeMAX_String_NUM+1) THEN
	error:=TRUE;
	errTxt:='dataBase$'s length too short';
	RETURN;
END_IF
IF csv_rows<(dataStringLength+1) THEN
	error:=TRUE;
	errTxt:='dataBase$'s length too short';
	RETURN;
END_IF


IF initB AND (NOT busy) THEN
	RETURN;
END_IF
initB:=TRUE;

//header
	pDatabase[0,0]:='NUM';//NUM
	pDatabase[0,1]:='RecipeID';//data type
	pDatabase[0,2]:='RecipeNAME';//name
	pDatabase[0,3]:='StepID';//value
	pDatabase[0,4]:='etchTime';//set
	pDatabase[0,5]:='rfPoint_source';//set
	pDatabase[0,6]:='pdvPoint';//set
	pDatabase[0,7]:='mfc1';//set
	pDatabase[0,8]:='mfc2';//set
	pDatabase[0,9]:='mfc3';//set
	pDatabase[0,10]:='mfc4';//set
	pDatabase[0,11]:='mfc5';//set
	pDatabase[0,12]:='mfc6';//set
	pDatabase[0,13]:='mfc7';//set
	pDatabase[0,14]:='mfc8';//set
	pDatabase[0,15]:='mfc9';//set
	pDatabase[0,16]:='rfPoint_Power';//set
	pDatabase[0,17]:='par_2';//set
	pDatabase[0,18]:='par_3';//set
	pDatabase[0,19]:='par_4';//set
	
(*--- 不在此处填充，转移到保存数据时填充
//bool
FOR i:=1 TO (dataBoolLength+1) DO
	//pDatabase[i,0]:=UDINT_TO_STRING(i-1);//NUM  --- 不在此处填充
	//pDatabase[i,1]:='BOOL';//data type --- 不在此处填充
	//pDatabase[i,2]:='';//name
	//pDatabase[i,3]:=BOOL_TO_STRING(FALSE);//value
	//pDatabase[i,4]:='';//no use
END_FOR

//dint
FOR i:=(dataBoolLength+2) TO (dataBoolLength+2+dataDintLength) DO
	//pDatabase[i,0]:=UDINT_TO_STRING(i-(dataBoolLength+2));//NUM  --- 不在此处填充
	//pDatabase[i,1]:='DINT';//data type --- 不在此处填充
	//pDatabase[i,2]:='';//name
	//pDatabase[i,3]:=DINT_TO_STRING(0);//value
	//pDatabase[i,4]:='';//no use
END_FOR

//lreal
FOR i:=(dataBoolLength+dataDintLength+3) TO (dataBoolLength+dataDintLength+dataLrealLength+3) DO
	//pDatabase[i,0]:=UDINT_TO_STRING(i-(dataBoolLength+dataDintLength+3));//NUM  --- 不在此处填充
	//pDatabase[i,1]:='LREAL';//data type --- 不在此处填充
	//pDatabase[i,2]:='';//name
	//pDatabase[i,3]:=DINT_TO_STRING(0);//value
	//pDatabase[i,4]:='';//no use
END_FOR
*)
END_METHOD

METHOD IsAllDigits  : BOOL
VAR_INPUT
    str : STRING(255); // 假设字符串最大长度为255
END_VAR
VAR
    i : INT;
    ch : BYTE;
END_VAR
IsAllDigits := TRUE; // 初始假设字符串全为数字

FOR i := 0 TO LEN(str)-1 DO
    ch := (str[i]);
    IF (ch < 48) OR (ch > 57) THEN
        IsAllDigits := FALSE; 
		EXIT;
    END_IF
END_FOR
END_METHOD

METHOD PRIVATE readMethod : BOOL
VAR_INPUT
END_VAR
CASE readStep OF
0:
	IF (readB OR (NOT startUPb)) AND (NOT busy) THEN
		readStep:=1;
		startUPb:=TRUE;//for first time, 
		readB:=FALSE;
		rDone:=FALSE;
		busy:=TRUE;
		error:=FALSE;
		errID:=0;
		errTxt:='';
		fbFileOpen(bExecute:= FALSE);
		checkFileExistError:=FALSE;
//		pDatabase:=pClearDatabase;
		//gShowNum:=0;
	END_IF
	
1:
	fbFileOpen(
		sNetId:= , 
		sPathName:= sFileName, 
		nMode:= FOPEN_MODEREAD, 
		ePath:= PATH_GENERIC, 
		bExecute:= TRUE, 
		tTimeout:= , 
		bBusy=> , 
		bError=> , 
		nErrId=> , 
		hFile=> hFile);
	IF NOT fbFileOpen.bBusy THEN
		IF fbFileOpen.bError THEN
			checkFileExistError:=TRUE;
		END_IF
		fbFileOpen(bExecute:= FALSE);
		readStep:=2;
	END_IF
	fbFileClose(bExecute:= FALSE);
2:
	fbFileClose(
		sNetId:= , 
		hFile:= hFile, 
		bExecute:= TRUE, 
		tTimeout:= , 
		bBusy=> , 
		bError=> , 
		nErrId=> );
	IF NOT fbFileClose.bBusy THEN
		IF checkFileExistError THEN
			readStep:=110;
		ELSE
			readStep:=11;
		END_IF
		fbFileClose(bExecute:= FALSE);
	END_IF

11:
	//read txt to Database
	readTxt(
		database:= pDatabase, 
		csv_rows:= csv_rows, 
		csv_columns:= csv_columns, 
		bRead:= TRUE, 
		sFileName:= sFileName);
	readStep:=12;

12:
	readTxt(
		database:= pDatabase, 
		csv_rows:= csv_rows, 
		csv_columns:= csv_columns, 
		bRead:= FALSE, 
		sFileName:= sFileName,
		Error=>error,
		nErrId=>errID);
		
	IF error THEN
		readStep:=110;
		RETURN;
	END_IF
	
	IF NOT readTxt.bBusy THEN
		readStep:=13;
	END_IF
	
13:
	string2Data();
	readStep:=100;
	
100:
	rDone:=TRUE;
	busy:=FALSE;
	error:=error;
	errID:=errID;
	errTxt:=errTxt;
	IF NOT readB THEN
		readStep:=0;
	END_IF	


110:
	rDone:=FALSE;
	busy:=FALSE;
	error:=TRUE;
	errID:=errID;
	errTxt:='read data fail';	
	IF NOT readB THEN
		readStep:=0;
	END_IF		
	
END_CASE
END_METHOD

ACTION RecipeChange:
IF NOT (gRecipeShowNameOld=gRecipeNameSelect[gRecipeSelectIndex1].Name) AND NOT busy AND saveActStep<10 THEN
	gRecipeShowNameNow:=gRecipeNameSelect[gRecipeSelectIndex1].Name;
	readB:=TRUE;
END_IF
gRecipeShowNameOld:=gRecipeNameSelect[gRecipeSelectIndex1].Name;
END_ACTION

ACTION saveActRun:
IF saveAct THEN
	saveAct:=FALSE;
	IF saveActStep<10 THEN
		saveActStep:=10;
	END_IF
END_IF
CASE saveActStep OF
	0:
		ton1(IN:=FALSE);;	
	10:
		gRecipeNameSelect[gRecipeSelectIndex1].Name:=gRecipeShowNameNow;
		saveActStep:=saveActStep+10;
	20:
		ton1(IN:= NOT ton1.Q, PT:=T#0.1S);
		IF ton1.Q THEN
			ton1(IN:=FALSE);
			saveActStep:=saveActStep+10;
		END_IF
	30:
		IF NOT DataSave.fbDataSaveModule_EX_recipename.busy THEN
			DataSave.fbDataSaveModule_EX_recipename.saveB:=TRUE;
			saveActStep:=saveActStep+10;	
		END_IF
		ton1(IN:=FALSE);
	40:
		ton1(IN:= NOT ton1.Q, PT:=T#0.1S);
		IF ton1.Q THEN
			ton1(IN:=FALSE);
			saveActStep:=saveActStep+10;
		END_IF
	50:
		IF NOT DataSave.fbDataSaveModule_EX_recipename.busy THEN
			DataSave.fbDataSaveModule_EX_recipename.readB:=TRUE;
			saveActStep:=saveActStep+10;	
		END_IF
		ton1(IN:=FALSE);
	60:
		IF NOT DataSave.fbDataSaveModule_EX_recipe.busy THEN
			DataSave.fbDataSaveModule_EX_recipe.saveB:=TRUE;
			saveActStep:=saveActStep+10;
		END_IF
		ton1(IN:=FALSE);
	70:
		ton1(IN:= NOT ton1.Q, PT:=T#0.1S);
		IF ton1.Q THEN
			ton1(IN:=FALSE);
			saveActStep:=saveActStep+10;
		END_IF
	80:
		IF NOT DataSave.fbDataSaveModule_EX_recipe.busy THEN
			DataSave.fbDataSaveModule_EX_recipe.readB:=TRUE;
			saveActStep:=saveActStep+10;
		END_IF
	90:
		saveActStep:=0;
END_CASE
END_ACTION

METHOD PRIVATE saveMethod : BOOL
VAR_INPUT
END_VAR
CASE saveStep OF
0:
	IF saveB AND (NOT busy) THEN
		saveStep:=1;
		saveB:=FALSE;
		busy:=TRUE;
		sDone:=FALSE;
		error:=FALSE;
		errID:=0;
		errTxt:='';
	END_IF

1:
	createDir();
	data2String();
	saveStep:=2;
	
2:
	csv_rows:=INT_TO_UDINT(gShowNum);
	writeTxt(
		database:= pDatabase, 
		csv_rows:= csv_rows, 
		csv_columns:= csv_columns, 
		bWrite:= TRUE, 
		sFileName:= sFileName,
		sFileNameOld:= sFileNameOld);	
	saveStep:=3;

3:
	csv_rows:=INT_TO_UDINT(gShowNum);
	writeTxt(
		database:= pDatabase, 
		csv_rows:= csv_rows, 
		csv_columns:= csv_columns, 
		bWrite:= FALSE, 
		sFileName:= sFileName,
		sFileNameOld:= sFileNameOld,
		Error=>error,
		nErrID=>errID);	
	
	IF error THEN
		saveStep:=110;
		RETURN;
	END_IF

	IF NOT writeTxt.bBusy THEN
		saveStep:=100;
	END_IF

100:
	busy:=FALSE;
	sDone:=TRUE;
	error:=error;
	errID:=errID;
	errTxt:=errTxt;

	IF NOT saveB THEN
		saveStep:=0;
	END_IF

110:
	busy:=FALSE;
	sDone:=FALSE;
	error:=TRUE;
	errID:=errID;
	errTxt:='save data fail';

	IF NOT saveB THEN
		saveStep:=0;
	END_IF
END_CASE
END_METHOD

METHOD setValue : BOOL
VAR_INPUT
	value:STRING;
END_VAR
VAR_INPUT
	rnum:UDINT;
	cnum:UDINT;
END_VAR
IF 0<=rnum AND rnum<=dataStringLength
	AND 0<=cnum AND cnum<=gRecipeMAX_CSV_COLUMNS THEN
	pDatabase[rnum,cnum]:=value;
	setValue:=TRUE;
ELSE
	setValue:=FALSE;
END_IF
END_METHOD

METHOD PRIVATE string2Data : BOOL
VAR_INPUT
END_VAR
VAR
	i:INT:=0;
	index_temp:UDINT;
END_VAR
//judge length
IF gRecipeMAX_CSV_ROWS<(gRecipeMAX_String_NUM+1) THEN
	error:=TRUE;
	errTxt:='dataBase$'s length too short';
	RETURN;
END_IF
IF csv_rows<(dataStringLength+1) THEN
	error:=TRUE;
	errTxt:='dataBase$'s length too short';
	RETURN;
END_IF

(*
//bool
FOR i:=0 TO dataBoolLength DO
	dataBool[i]:=STRING_TO_BOOL(pDatabase[i+1,3]);//value
END_FOR

//dint
FOR i:=(dataBoolLength+1) TO (dataBoolLength+1+dataDintLength) DO
	dataDint[i-(dataBoolLength+1)]:=STRING_TO_DINT(pDatabase[i+1,3]);//value
END_FOR

//lreal
FOR i:=(dataBoolLength+dataDintLength+2) TO (dataBoolLength+dataDintLength+dataLrealLength+2) DO
	dataLreal[i-(dataBoolLength+dataDintLength+2)]:=STRING_TO_LREAL(pDatabase[i+1,3]);//value
END_FOR
*)
FOR i:=0 TO UDINT_TO_INT(gRecipeMAX_CSV_ROWS) DO
	dataString[i,0]:=(pDatabase[i,0]);
	dataString[i,1]:=(pDatabase[i,1]);
	dataString[i,2]:=(pDatabase[i,2]);
	dataString[i,3]:=(pDatabase[i,3]);
	dataString[i,4]:=(pDatabase[i,4]);
	dataString[i,5]:=(pDatabase[i,5]);
	dataString[i,6]:=(pDatabase[i,6]);
	dataString[i,7]:=(pDatabase[i,7]);
	dataString[i,8]:=(pDatabase[i,8]);
	dataString[i,9]:=(pDatabase[i,9]);
	dataString[i,10]:=(pDatabase[i,10]);
	dataString[i,11]:=(pDatabase[i,11]);
	dataString[i,12]:=(pDatabase[i,12]);
	dataString[i,13]:=(pDatabase[i,13]);
	dataString[i,14]:=(pDatabase[i,14]);
	dataString[i,15]:=(pDatabase[i,15]);
	dataString[i,16]:=(pDatabase[i,16]);
	dataString[i,17]:=(pDatabase[i,17]);
	dataString[i,18]:=(pDatabase[i,18]);
	dataString[i,19]:=(pDatabase[i,19]);
	
	IF (pDatabase[i+1,2]=gRecipeShowNameNow) AND NOT (pDatabase[i+1,4]='') AND NOT (pDatabase[i+1,5]='') AND NOT (pDatabase[i+1,6]='') AND
	NOT (pDatabase[i+1,7]='') AND NOT (pDatabase[i+1,8]='') AND NOT (pDatabase[i+1,9]='') AND NOT (pDatabase[i+1,10]='') AND
	NOT (pDatabase[i+1,11]='') AND NOT (pDatabase[i+1,12]='') AND NOT (pDatabase[i+1,13]='') AND NOT (pDatabase[i+1,14]='') AND
	NOT (pDatabase[i+1,15]='') AND NOT (pDatabase[i+1,16]='') AND NOT (pDatabase[i+1,17]='') AND NOT (pDatabase[i+1,18]='') THEN
		gRecipeEditorData[i+1].NUM:=(pDatabase[i+1,0]);
		gRecipeEditorData[i+1].etchTime:=(pDatabase[i+1,4]);
		gRecipeEditorData[i+1].rfPoint_source:=(pDatabase[i+1,5]);
		gRecipeEditorData[i+1].pdvPoint:=(pDatabase[i+1,6]);
		gRecipeEditorData[i+1].mfc1:=(pDatabase[i+1,7]);
		gRecipeEditorData[i+1].mfc2:=(pDatabase[i+1,8]);
		gRecipeEditorData[i+1].mfc3:=(pDatabase[i+1,9]);
		gRecipeEditorData[i+1].mfc4:=(pDatabase[i+1,10]);
		gRecipeEditorData[i+1].mfc5:=(pDatabase[i+1,11]);
		gRecipeEditorData[i+1].mfc6:=(pDatabase[i+1,12]);
		gRecipeEditorData[i+1].mfc7:=(pDatabase[i+1,13]);
		gRecipeEditorData[i+1].mfc8:=(pDatabase[i+1,14]);
		gRecipeEditorData[i+1].mfc9:=(pDatabase[i+1,15]);
		gRecipeEditorData[i+1].rfPoint_Power:=(pDatabase[i+1,16]);
		gRecipeEditorData[i+1].par_2:=(pDatabase[i+1,17]);
		gRecipeEditorData[i+1].par_3:=(pDatabase[i+1,18]);
		gRecipeEditorData[i+1].par_4:=(pDatabase[i+1,19]);
		IF LEN(gRecipeEditorData[i+1].NUM)=0 AND (i+1<>UDINT_TO_INT(gRecipeMAX_CSV_ROWS)) THEN
			gShowNum:=i;
			gRecipeViewData:=gRecipeEditorData;
			RETURN;
		END_IF
	ELSE
		gShowNum:=i;
		gRecipeViewData:=gRecipeEditorData;
		RETURN;
	END_IF
	
	
	
END_FOR
END_METHOD

ACTION VersionLog:
(*
版本: V1.0.0.0 20241012  CPH
说明:
	1. 首个版本
(**************************************************)
版本: V1.0.0.1
说明:
	1. 增加参数备份文件，文件名以原文件名+时间命名
(**************************************************)
*)
END_ACTION

END_FUNCTION_BLOCK

// ---- POUs/BaseModule/DataSaveModule_EX/csvReadWriteInTextMode/P_TextModeWrite_Recipe.TcPOU
FUNCTION_BLOCK P_TextModeWrite_Recipe
VAR_IN_OUT
	database		: ARRAY[0..gRecipeMAX_CSV_ROWS, 0..gRecipeMAX_CSV_COLUMNS ] OF STRING(30);
	csv_rows		: UDINT;
	csv_columns		: UDINT;
END_VAR
VAR_INPUT
	bWrite			: BOOL := FALSE;(* Rising edge starts program execution *)	
	sFileName		: T_MaxString := '';(* CSV destination file path and name *)
	sFileNameOld	:T_MaxString := '';(*旧文件名*)
END_VAR
VAR_OUTPUT
	bBusy			: BOOL;
	error			: BOOL;
	nErrId			: UDINT;	
END_VAR
VAR
	bError			: BOOL;
	sNetId			: T_AmsNetId := '';	(* TwinCAT system network address *)

	sCSVLine		: T_MaxString := '';(* Single CSV text line (row, record), we are using string as record buffer (your are able to see created fields) *)
	sCSVField		: T_MaxString := '';(* Single CSV field value (column, record field) *)
	//sCSVField		: UDINT;

	nRow	 		: UDINT 	:= 0;(* Row number (record) *)
	nColumn			: UDINT 	:= 0;(* Column number (record field) *)
	hFile			: UINT		:= 0;(* File handle of the source file *)
	step			: DWORD 	:= 0;
	fbFileOpen		: FB_FileOpen;(* Opens file *)
	fbFileClose		: FB_FileClose;(* Closes file *)
	fbFilePuts		: FB_FilePuts;(* Writes one record (line) *)
	fbFileWrite     : FB_FileWrite;
	fbWriter		: FB_CSVMemBufferWriter;(* Helper function block used to create CSV data bytes (single record line) *)
    StringModelWrite		: StringModel_256000_EX;
	fbFileRename			: FB_FileRename;//修改文件名称
	fbFileDelete			: FB_FileDelete;//删除文件
	writeTON				: TON;//延时写入

	(* :=[ (* Source PLC database *)
	'0_0', '0_1', '0_2', '0_3', '0_4', '0_5',
	'1_0', '1_1', '1_2', '1_3', '1_4', '1_5',
	'2_0', '2_1', '2_2', '2_3', '2_4', '2_5',
	'3_0', '3_1', '3_2', '3_3', '3_4', '3_5',
	'4_0', '4_1', '4_2', '4_3', '4_4', '4_5',
	'5_0', '5_1', '5_2', '5_3', '5_4', '5_5'];*)

END_VAR

DEFAULT_CSV_FIELD_SEP:= 16#2C;  //配置CSV文件的分割符，16#2C表明各个参数之间是用逗号分隔的。
CASE step OF
	0:(* Wait for rising edge at bWrite variable *)
		IF bWrite THEN
			bWrite 	:= FALSE;
			bBusy 	:= TRUE;
			error	:= FALSE;
			bError	:= FALSE;
			nErrId	:= 0;
			hFile	:= 0;
			nRow	:= 0;
			nColumn	:= 0;
			step 	:= 1;
		END_IF
	1:
		StringModelWrite.init();
		fbFileDelete(bExecute:= FALSE);
		fbFileRename(bExecute:= FALSE);
		step:=2;
	2:
		fbFileDelete(
			sNetId:= , 
			sPathName:= sFileNameOld, 
			ePath:= PATH_GENERIC, 
			bExecute:= TRUE, 
			tTimeout:= DEFAULT_ADS_TIMEOUT, 
			bBusy=> , 
			bError=> , 
			nErrId=> );
		step:=3;
	3:
		fbFileDelete(bExecute:= FALSE);
		IF NOT fbFileDelete.bBusy THEN
			step:=4;
		END_IF
	4:
		fbFileRename(
			sNetId:= , 
			sOldName:= sFileName, 
			sNewName:= sFileNameOld, 
			ePath:= PATH_GENERIC, 
			bExecute:= TRUE, 
			tTimeout:= DEFAULT_ADS_TIMEOUT, 
			bBusy=> , 
			bError=> , 
			nErrId=> );
		step:=5;
	5:
		fbFileRename(bExecute:= FALSE);
		IF NOT fbFileRename.bBusy THEN
			step:=10;
		END_IF

	10:(* Open source file *)
		fbFileOpen(  bExecute := FALSE  );
		fbFileOpen( sNetId := sNetId, sPathName := sFileName, nMode := FOPEN_MODEWRITE OR FOPEN_MODETEXT,(* Open file in TEXT mode! *)
					ePath := PATH_GENERIC, bExecute := TRUE );
		step := 20;

	20:(* Wait until open not busy *)
		//StringModelWrite.init();
		fbFileOpen( bExecute := FALSE, bError => bError, nErrID => nErrID, hFile => hFile );
		IF NOT fbFileOpen.bBusy THEN
			IF NOT fbFileOpen.bError THEN
				step := 30;
			ELSE(* Error: file not found? *)
				step := 1000;
			END_IF
		END_IF
	
	30:(* Convert one PLC record to CSV format *)
		FOR nRow:=0 TO csv_rows BY 1 DO
				sCSVLine := '';
				fbWriter.eCmd := eEnumCmd_First;(* Write first field value *)
			FOR nColumn := 0 TO csv_columns BY 1 DO
				sCSVField := STRING_TO_CSVFIELD( database[ nRow, nColumn ], FALSE );(* TODO: Get field value from your application *)
				(* Add new field to the record buffer *)
				fbWriter( 	pBuffer := ADR( sCSVLine ), cbBuffer := SIZEOF( sCSVLine ) - 1, putValue := sCSVField, pValue := 0, cbValue := 0,
							bCRLF := ( nColumn = csv_columns ) );(* bCRLF == TRUE => Write CRLF after the last field value *)
				IF fbWriter.bOk THEN
					fbWriter.eCmd := eEnumCmd_Next;(* Write next field value *)
				ELSE(* Error *)
					step := 1000;
					RETURN;
				END_IF
			END_FOR
			(* FB_FilePuts adds allready CR (carriage return) to the written line.
			We have to replace the $R$L characters with $L character to avoid double CR. *)
			IF RIGHT( sCSVLine, 2 ) = '$R$L' THEN
				sCSVLine := REPLACE( sCSVLine, '$L', 2, LEN( sCSVLine ) - 1 );
			END_IF
            StringModelWrite.append(str:= sCSVLine);
		END_FOR
		IF nRow> csv_rows THEN
			step := 40;(* Write record to the file *)
		END_IF
		writeTON(IN:=FALSE);

	40:(* Write record to file *)
		fbFileWrite( bExecute := FALSE );
		writeTON(IN:=NOT writeTON.Q,PT:=T#50MS);
		IF writeTON.Q THEN
			//fbFileWrite( sNetId := sNetId, hFile := hFile, pWriteBuff := StringModelWrite.getAddr, cbWriteLen := StringModelWrite.length, bExecute := TRUE );
			fbFileWrite( sNetId := sNetId, hFile := hFile, pWriteBuff := ADR(StringModelWrite.b), cbWriteLen := StringModelWrite.length, bExecute := TRUE );
			step := 50;
		END_IF

	50:(* Wait until write not busy *)
		fbFileWrite( bExecute := FALSE, bError => bError, nErrID => nErrID );
		IF NOT fbFileWrite.bBusy THEN
			IF NOT fbFileWrite.bError THEN
				step := 100;(* Write next record *)
			ELSE(* Error *)
				step := 1000;
			END_IF
		END_IF
		
	100:(* Close source file *)
		fbFileClose( bExecute := FALSE );
		fbFileClose( sNetId := sNetId, hFile := hFile, bExecute := TRUE );
		step := 110;

	110:(* Wait until close not busy *)
		fbFileClose( bExecute := FALSE, bError => bError, nErrID => nErrID );
		IF NOT fbFileClose.bBusy THEN
			hFile := 0;
			step := 1000;
		END_IF

	1000:(* Error or ready step => cleanup *)
		IF ( hFile <> 0 ) THEN
			step := 100; (* Close the source file *)
		ELSE
			bBusy := FALSE;
			error := bError;
			step := 0;	(* Ready *)
		END_IF
END_CASE

END_FUNCTION_BLOCK

// ---- POUs/BaseModule/DataSaveModule_EX/csvReadWriteInTextMode/P_TextModeRead_Recipe.TcPOU
FUNCTION_BLOCK P_TextModeRead_Recipe
VAR_IN_OUT
	database		: ARRAY[0..gRecipeMAX_CSV_ROWS, 0..gREcipeMAX_CSV_COLUMNS ] OF STRING(30);(* Target PLC database *)
	csv_rows		: UDINT;
	csv_columns		: UDINT;
END_VAR
VAR_INPUT
	bRead			: BOOL := FALSE;(* Rising edge starts program execution *)	
	sFileName		: T_MaxString := '';(* CSV source file path and name *)
END_VAR
VAR_OUTPUT
	bBusy			: BOOL;
	error			: BOOL;
	nErrId			: UDINT;	
END_VAR
VAR
	bError			: BOOL;
	readData:ARRAY[gNumBegin..(gMaxNumLength+gNumBegin-1)]OF BYTE;
	readDataClear:ARRAY[gNumBegin..(gMaxNumLength+gNumBegin-1)]OF BYTE;
	sNetId			: T_AmsNetId := '';	(* TwinCAT system network address *)
	sCSVLine		: T_MaxString := '';(* Single CSV text line (row, record), we are using string as record buffer (your are able to see read fields)  *)
	sCSVField		: T_MaxString := '';(* Single CSV field value (column, record field) *)
	nRow	 		: UDINT 	:= 0;(* Row number (record) *)
	nColumn			: UDINT 	:= 0;(* Column number (record field) *)
	hFile			: UINT		:= 0;(* File handle of the source file *)
	step			: DWORD 	:= 0;
	fbFileOpen		: FB_FileOpen;(* Opens file *)
	fbFileClose		: FB_FileClose;(* Closes file *)
	fbFileGets		: FB_FileGets;(* Reads one record (line) *)
	fbFileRead		: FB_FileRead;//---------------------------------------
	fbReader		: FB_CSVMemBufferReader;(* Helper function block used to parse CSV data bytes (single record line) *)

	strTemp : T_MaxString;
	strT : T_MaxString;
	i : UDINT:=0;
	iTemp : UDINT:=0;
END_VAR

DEFAULT_CSV_FIELD_SEP:= 16#2C;  //配置CSV文件的分割符，16#2C表明各个参数之间是用逗号分隔的。
CASE step OF
	0:	(* Wait for rising edge at bRead variable *)
		IF bRead THEN
			bRead 	:= FALSE;
			bBusy 	:= TRUE;
			error:= bError	:= FALSE;
			nErrId	:= 0;
			hFile	:= 0;
			nRow	:= 0;
			nColumn	:= 0;
			MEMSET( ADR( database ), 0, SIZEOF( database ) );
			step 		:= 1;
			readData:=readDataClear;
		END_IF

	1:	(* Open source file *)
		fbFileOpen(  bExecute := FALSE  );
		fbFileOpen( sNetId := sNetId, sPathName := sFileName, nMode := FOPEN_MODEREAD OR FOPEN_MODETEXT,(* Open file in TEXT mode! *)
					ePath := PATH_GENERIC, bExecute := TRUE );
		step := 2;

	2:(* Wait until open not busy *)
		fbFileOpen( bExecute := FALSE, bError => bError, nErrID => nErrID, hFile => hFile );
		IF NOT fbFileOpen.bBusy THEN
			IF NOT fbFileOpen.bError THEN
				step := 3;
			ELSE(* Error: file not found? *)
				step := 100;
			END_IF
		END_IF
		
	3:
		step := 4;
	4:
		fbFileRead(
			sNetId:= sNetId, 
			hFile:= hFile, 
			bExecute:= FALSE,);
		step := 5;
	5:(*Read data from file*)
		fbFileRead(
			sNetId:= sNetId, 
			hFile:= hFile, 
			pReadBuff:= ADR(readData),
			cbReadLen:= gMaxNumLength,
			bExecute:= TRUE, 
			tTimeout:= , 
			bBusy=> , 
			bError=> , 
			nErrId=> , 
			cbRead=> , 
			bEOF=> );
		IF NOT fbFileRead.bBusy AND NOT fbFileRead.bError THEN
			IF fbFileRead.bEOF THEN
				step := 6;
			END_IF
			step := 6;
			fbFileRead(
				sNetId:= sNetId, 
				hFile:= hFile, 
				bExecute:= FALSE,);
		ELSIF fbFileRead.bError THEN
			step := 100;
		END_IF
		sCSVLine := '';
		iTemp:=1;
	6:
		FOR nRow:=0 TO csv_rows BY 1 DO
			sCSVLine := '';
			FOR i:=iTemp TO gMaxNumLength BY 1 DO
				strT := F_ToCHR(c:=readData[i]);
				IF '$L' = strT THEN
					strTemp:=CONCAT(STR1:=sCSVLine,STR2:='$R$L');
					iTemp:=i+1;
					EXIT;
				ELSE
					sCSVLine:=CONCAT(STR1:=sCSVLine,STR2:=strT);
				END_IF
			END_FOR
			fbReader.eCmd := eEnumCmd_First;(* Read first field value *)
			FOR nColumn := 0 TO csv_columns BY 1 DO
				fbReader( pBuffer := ADR( sCSVLine ), cbBuffer := SIZEOF( sCSVLine ), getValue => sCSVField);
				IF fbReader.bOk THEN
					fbReader.eCmd := eEnumCmd_Next;
					IF ( nRow <= csv_rows ) THEN
						IF ( nColumn <= csv_columns ) THEN
							database[nRow, nColumn] := CSVFIELD_TO_STRING( sCSVField, FALSE );
						END_IF
					END_IF
				END_IF
			END_FOR
			IF fbReader.bCRLF THEN(* CRLF == TRUE => End of reacord reached *)
				nColumn := 0;
			END_IF
		END_FOR
		step := 10;

	10:	(* Close source file *)
		fbFileClose( bExecute := FALSE );
		fbFileClose( sNetId := sNetId, hFile := hFile, bExecute := TRUE );
		step := 11;

	11:(* Wait until close not busy *)
		fbFileClose( bExecute := FALSE, bError => bError, nErrID => nErrID );
		IF ( NOT fbFileClose.bBusy ) THEN
			hFile := 0;
			step := 100;
		END_IF

	100: (* Error or ready step => cleanup *)
		IF ( hFile <> 0 ) THEN
			step := 10; (* Close the source file *)
		ELSE
			bBusy := FALSE;
			error := bError;
			step := 0;	(* Ready *)
		END_IF

END_CASE

END_FUNCTION_BLOCK

// ---- POUs/BaseModule/DataSaveModule_EX/csvReadWriteInTextMode/P_TextModeDelete_1.TcPOU
FUNCTION_BLOCK P_TextModeDelete_1
VAR_INPUT
	bDelete			: BOOL := FALSE;(* Rising edge starts program execution *)	
	sFileName		: T_MaxString := '';(* CSV destination file path and name *)
	sFileNameOld	:T_MaxString := '';(*旧文件名*)
END_VAR
VAR_OUTPUT
	bBusy			: BOOL;
	error			: BOOL;
	nErrId			: UDINT;	
END_VAR
VAR
	bError			: BOOL;
	sNetId			: T_AmsNetId := '';	(* TwinCAT system network address *)

	sCSVLine		: T_MaxString := '';(* Single CSV text line (row, record), we are using string as record buffer (your are able to see created fields) *)
	sCSVField		: T_MaxString := '';(* Single CSV field value (column, record field) *)
	//sCSVField		: UDINT;

	nRow	 		: UDINT 	:= 0;(* Row number (record) *)
	nColumn			: UDINT 	:= 0;(* Column number (record field) *)
	hFile			: UINT		:= 0;(* File handle of the source file *)
	step			: DWORD 	:= 0;
	fbFileOpen		: FB_FileOpen;(* Opens file *)
	fbFileClose		: FB_FileClose;(* Closes file *)
	fbFilePuts		: FB_FilePuts;(* Writes one record (line) *)
	fbFileWrite     : FB_FileWrite;
	fbFileDelete	: FB_FileDelete;// 文档删除
	fbWriter		: FB_CSVMemBufferWriter;(* Helper function block used to create CSV data bytes (single record line) *)
    StringModelWrite		: StringModel_256000_EX;
	fbFileRename			: FB_FileRename;//修改文件名称
	writeTON				: TON;//延时写入

	(* :=[ (* Source PLC database *)
	'0_0', '0_1', '0_2', '0_3', '0_4', '0_5',
	'1_0', '1_1', '1_2', '1_3', '1_4', '1_5',
	'2_0', '2_1', '2_2', '2_3', '2_4', '2_5',
	'3_0', '3_1', '3_2', '3_3', '3_4', '3_5',
	'4_0', '4_1', '4_2', '4_3', '4_4', '4_5',
	'5_0', '5_1', '5_2', '5_3', '5_4', '5_5'];*)

END_VAR

DEFAULT_CSV_FIELD_SEP:= 16#2C;  //配置CSV文件的分割符，16#2C表明各个参数之间是用逗号分隔的。
CASE step OF
	0:(* Wait for rising edge at bWrite variable *)
		IF bDelete THEN
			bDelete 	:= FALSE;
			bBusy 	:= TRUE;
			error	:= FALSE;
			bError	:= FALSE;
			nErrId	:= 0;
			hFile	:= 0;
			nRow	:= 0;
			nColumn	:= 0;
			step 	:= 1;
		END_IF
	1:
		StringModelWrite.init();
		fbFileDelete(bExecute:= FALSE);
		fbFileRename(bExecute:= FALSE);
		step:=2;
	2:
		fbFileDelete(
			sNetId:= , 
			sPathName:= sFileName, 
			ePath:= PATH_GENERIC, 
			bExecute:= TRUE, 
			tTimeout:= DEFAULT_ADS_TIMEOUT, 
			bBusy=> , 
			bError=> , 
			nErrId=> );
		step:=3;
	3:
		fbFileDelete(bExecute:= FALSE);
		IF NOT fbFileDelete.bBusy THEN
			step:=4;
		END_IF
	4:
		step:=1000;

	1000:(* Error or ready step => cleanup *)
		IF ( hFile <> 0 ) THEN
			step := 100; (* Close the source file *)
		ELSE
			bBusy := FALSE;
			error := bError;
			step := 0;	(* Ready *)
		END_IF
END_CASE

END_FUNCTION_BLOCK

// ---- POUs/BaseModule/Error/error_Trigger.TcPOU
//设备报警处理
FUNCTION error_Trigger : BOOL
VAR_INPUT
	errorID					:DINT;//error id
END_VAR
VAR
END_VAR

IF g_Max_Data_Elements<=gError_hTable.nCount THEN//哈希表内容超过100条，直接返回
	RETURN;
END_IF
gError_fbTable.A_Lookup(key:=TO_DWORD(errorID),hTable:=gError_hTable);//从哈希表中查询是否有正在报警的id
IF gError_fbTable.bOk THEN//如果有，直接返回，不再报警该id；如果无，则添加到哈希表中，并报警提示
	//value:= gError_fbTable.getValue;
	RETURN;//已经报警过该错误
ELSE
	(* Entry not found *)
	gError_fbTable.A_Add(key:=TO_DWORD(errorID),putValue :=TO_UDINT(errorID), hTable:=gError_hTable);
END_IF
//print之前，先进行ErrorMonitor将错误内容进行分配；如果错误内容写死，可以不用这么写
errorMonitor();
error_Printf(errorID);

IF g_d_ErrorBegin<=errorID AND errorID<=g_d_ErrorEnd THEN
	CASE gErrorARRAY[errorID].eErrLevel OF
		Error_Level_0:
			//gErrorARRAY[errorID].bError:=TRUE;
			IF gAutoRunningFlag THEN
				//PLC_MainSW.appendSend(0,0,E_CmdID_SW.SW_Error,0.0,0.0,0.0,0.0,gErrorARRAY[errorID].eErrLevel,gErrorARRAY[errorID].uErrID,gErrorARRAY[errorID].sErrTXT);
				//PLC_MainSW.appendSend(0,0,E_CmdID_SW.SW_Error,0.0,0.0,0.0,0.0,0.0,ErrCodeProcess(errorID),'');
				//PLC_MainSW.appendSend(TO_STRING(ErrCodeProcess(errorID)));
			END_IF
		Error_Level_1:
			//gErrorARRAY[errorID].bError:=TRUE;
			IF gAutoRunningFlag THEN
				//PLC_MainSW.appendSend(0,0,E_CmdID_SW.SW_Error,0.0,0.0,0.0,0.0,gErrorARRAY[errorID].eErrLevel,gErrorARRAY[errorID].uErrID,gErrorARRAY[errorID].sErrTXT);
				//PLC_MainSW.appendSend(TO_STRING(ErrCodeProcess(errorID)));
			END_IF
		Error_Level_2:
			//gErrorARRAY[errorID].bError:=TRUE;
			IF gAutoRunningFlag THEN
				//PLC_MainSW.appendSend(0,0,E_CmdID_SW.SW_Error,0.0,0.0,0.0,0.0,gErrorARRAY[errorID].eErrLevel,gErrorARRAY[errorID].uErrID,gErrorARRAY[errorID].sErrTXT);
				//PLC_MainSW.appendSend(TO_STRING(ErrCodeProcess(errorID)));
			END_IF
		Error_Level_3:
			gErrorARRAY[errorID].bError:=TRUE;
			IF gAutoRunningFlag THEN
				//PLC_MainSW.appendSend(0,0,E_CmdID_SW.SW_Error,0.0,0.0,0.0,0.0,gErrorARRAY[errorID].eErrLevel,gErrorARRAY[errorID].uErrID,gErrorARRAY[errorID].sErrTXT);
				//PLC_MainSW.appendSend(TO_STRING(ErrCodeProcess(errorID)));
			END_IF
		Error_Level_4:
			gErrorARRAY[errorID].bError:=TRUE;
			IF gAutoRunningFlag THEN
				//PLC_MainSW.appendSend(0,0,E_CmdID_SW.SW_Error,0.0,0.0,0.0,0.0,gErrorARRAY[errorID].eErrLevel,gErrorARRAY[errorID].uErrID,gErrorARRAY[errorID].sErrTXT);
				//PLC_MainSW.appendSend(TO_STRING(ErrCodeProcess(errorID)));
			END_IF
	END_CASE
END_IF

END_FUNCTION

// ---- POUs/BaseModule/Error/errorMonitor.TcPOU
PROGRAM errorMonitor
VAR
	baseErrID:LINT;

	iTempInit:DINT:=0;
	bInit:BOOL;
	swStopMsg:wstring;
END_VAR
VAR
	cy_index_LRobot:INT;
	cy_index_Test:INT;
	cy_index_Buff:INT;
	cy_index_BIN1:INT;
	cy_index_BIN2:INT;
	cy_index_ULRobot:INT;
	
	bInit_Axis:BOOL;
	nInit_Axis:UINT;
	pAxisArr:ARRAY [1..nMaxNum_Axis] OF POINTER TO FB_MotorMovements;
	r_trig_AxisArr:ARRAY [1..nMaxNum_Axis] OF R_TRIG;
	nTemp_Axis:UINT;
	
	r_trig_RobotArr:ARRAY [1..2] OF R_TRIG;
	
	bInit_Cy:BOOL;
	nInit_Cy:UINT;
	pCyArr:ARRAY [1..nMaxNum_Cy] OF POINTER TO CylinderModule;
	r_trig_CyArr:ARRAY [1..nMaxNum_Cy] OF R_TRIG;
	nTemp_Cy:UINT;
	
	bInit_MFC:BOOL;
	nInit_MFC:UINT;
	pMFCArr:ARRAY [1..nMaxNum_MFC] OF POINTER TO MFCModule;
	r_trig_MFCArr:ARRAY [1..nMaxNum_MFC] OF R_TRIG;
	nTemp_MFC:UINT;
	
	bInit_TMP:BOOL;
	nInit_TMP:UINT;
	pTMPArr:ARRAY [1..nMaxNum_Vpe] OF POINTER TO TMPModule;
	r_trig_TMPArr:ARRAY [1..nMaxNum_TMP] OF R_TRIG;
	nTemp_TMP:UINT;
	
	bInit_Vpe:BOOL;
	nInit_Vpe:UINT;
	pVpeArr:ARRAY [1..nMaxNum_Vpe] OF POINTER TO VPEModule;
	r_trig_VpeArr:ARRAY [1..nMaxNum_Vpe] OF R_TRIG;
	nTemp_Vpe:UINT;
	
	bInit_PDV:BOOL;
	nInit_PDV:UINT;
	pPDVArr:ARRAY [1..nMaxNum_PDV] OF POINTER TO PVModule;
	r_trig_PDVArr:ARRAY [1..nMaxNum_PDV] OF R_TRIG;
	nTemp_PDV:UINT;
	
	bInit_RF:BOOL;
	nInit_RF:UINT;
	pRFArr:ARRAY [1..nMaxNum_RF] OF POINTER TO RFModule;
	r_trig_RFArr:ARRAY [1..nMaxNum_RF] OF R_TRIG;
	nTemp_RF:UINT;
	
	bInit_Chiller:BOOL;
	nInit_Chiller:UINT;
	pChillerArr:ARRAY [1..nMaxNum_Chiller] OF POINTER TO ChillerModule_1;
	r_trig_ChillerArr:ARRAY [1..nMaxNum_Chiller] OF R_TRIG;
	nTemp_Chiller:UINT;
	
	bInit_ARM:BOOL;
	nInit_ARM:UINT;
	pARMArr:ARRAY [1..nMaxNum_ARM] OF POINTER TO ARMModule;
	r_trig_ARMArr:ARRAY [1..nMaxNum_Chiller] OF R_TRIG;
	nTemp_ARM:UINT;
END_VAR
VAR CONSTANT
	nMaxNum_Axis:UINT:=100;
	nMaxNum_Cy:UINT:=200;
	nMaxNum_MFC:UINT:=20;
	nMaxNum_Vpe:UINT:=10;
	nMaxNum_TMP:UINT:=10;
	nMaxNum_PDV:UINT:=10;
	nMaxNum_RF:UINT:=10;
	nMaxNum_Chiller:UINT:=2;
	nMaxNum_ARM:UINT:=1;
END_VAR

IF NOT bInit THEN
	bInit:=TRUE;
	F_CreateHashTableHnd(ADR(gError_table),SIZEOF(gError_table),gError_hTable);(* Intialize table handle *)
END_IF


(* 此处是用于设备报错信息、报错ID的分配以及上报 *)
baseErrID:=0;// 通过改变变量值可实现 error ID的基础值

FOR iTempInit:=g_d_ErrorBegin TO g_d_ErrorEnd DO
	gErrorARRAY[iTempInit].uErrID:=baseErrID+iTempInit;// Error ID 分配
	IF gErrorARRAY[iTempInit].bError THEN
		gRunningState:=RunningStatus.eErrorState;// 进入Error状态
	END_IF
	IF gErrorARRAY[iTempInit].eErrLevel=4 THEN//用错误等级区分两个机台，从而实现两个机台的报警独立控制
		;
	END_IF
END_FOR
IF RunningStatus.eErrorState<>gRunningState THEN
	gErrTxtShow:='';
	gErrWTxtShow:=" ";
END_IF

(*
---------------------------------------------------------------------
*)

// error_Trigger(1);// 报警触发方式 示例
//////////////////////////////////////////////////////////////////////////////////////////////////1-20 严重错误,需重新回原
gErrorARRAY[0].eErrLevel:=Error_Level_1;// Error Level 分配
gErrorARRAY[0].sErrTXT:='This is a test message!';// Error 信息 分配
gErrorARRAY[0].sErrWTXT:=" 这是一个测试信息！";// Error 信息 分配

gErrorARRAY[1].eErrLevel:=Error_Level_4;// Error Level 分配
gErrorARRAY[1].sErrTXT:='E_Stop error!';// Error 信息 分配
gErrorARRAY[1].sErrWTXT:=" 急停错误！";// Error 信息 分配

gErrorARRAY[5].eErrLevel:=Error_Level_4;// Error Level 分配
gErrorARRAY[5].sErrTXT:='Slave device disconnected.';// Error 信息 分配
gErrorARRAY[5].sErrWTXT:=" 有从站设备掉线，请排除硬件问题后整机回原点";// Error 信息 分配


gErrorARRAY[10].eErrLevel:=Error_Level_4;// Error Level 分配
gErrorARRAY[10].sErrTXT:='Par etchTime input error.';// Error 信息 分配
gErrorARRAY[10].sErrWTXT:=" 输入的参数etchTime有误";// Error 信息 分配

gErrorARRAY[11].eErrLevel:=Error_Level_4;// Error Level 分配
gErrorARRAY[11].sErrTXT:='Par rfPoint_Source input error.';// Error 信息 分配
gErrorARRAY[11].sErrWTXT:=" 输入的参数rfPoint_Source有误";// Error 信息 分配

gErrorARRAY[12].eErrLevel:=Error_Level_4;// Error Level 分配
gErrorARRAY[12].sErrTXT:='Par pdvPoint input error.';// Error 信息 分配
gErrorARRAY[12].sErrWTXT:=" 输入的参数pdvPoint有误";// Error 信息 分配

gErrorARRAY[13].eErrLevel:=Error_Level_4;// Error Level 分配
gErrorARRAY[13].sErrTXT:='Par mfc1 input error.';// Error 信息 分配
gErrorARRAY[13].sErrWTXT:=" 输入的参数mfc1有误";// Error 信息 分配

gErrorARRAY[14].eErrLevel:=Error_Level_4;// Error Level 分配
gErrorARRAY[14].sErrTXT:='Par mfc2 input error.';// Error 信息 分配
gErrorARRAY[14].sErrWTXT:=" 输入的参数mfc2有误";// Error 信息 分配

gErrorARRAY[15].eErrLevel:=Error_Level_4;// Error Level 分配
gErrorARRAY[15].sErrTXT:='Par mfc3 input error.';// Error 信息 分配
gErrorARRAY[15].sErrWTXT:=" 输入的参数mfc3有误";// Error 信息 分配

gErrorARRAY[16].eErrLevel:=Error_Level_4;// Error Level 分配
gErrorARRAY[16].sErrTXT:='Par mfc4 input error.';// Error 信息 分配
gErrorARRAY[16].sErrWTXT:=" 输入的参数mfc4有误";// Error 信息 分配

gErrorARRAY[17].eErrLevel:=Error_Level_4;// Error Level 分配
gErrorARRAY[17].sErrTXT:='Par mfc5 input error.';// Error 信息 分配
gErrorARRAY[17].sErrWTXT:=" 输入的参数mfc5有误";// Error 信息 分配

gErrorARRAY[18].eErrLevel:=Error_Level_4;// Error Level 分配
gErrorARRAY[18].sErrTXT:='Par mfc6 input error.';// Error 信息 分配
gErrorARRAY[18].sErrWTXT:=" 输入的参数mfc6有误";// Error 信息 分配

gErrorARRAY[19].eErrLevel:=Error_Level_4;// Error Level 分配
gErrorARRAY[19].sErrTXT:='Par mfc7 input error.';// Error 信息 分配
gErrorARRAY[19].sErrWTXT:=" 输入的参数mfc7有误";// Error 信息 分配

gErrorARRAY[20].eErrLevel:=Error_Level_4;// Error Level 分配
gErrorARRAY[20].sErrTXT:='Par mfc8 input error.';// Error 信息 分配
gErrorARRAY[20].sErrWTXT:=" 输入的参数mfc8有误";// Error 信息 分配

gErrorARRAY[21].eErrLevel:=Error_Level_4;// Error Level 分配
gErrorARRAY[21].sErrTXT:='Par mfc9 input error.';// Error 信息 分配
gErrorARRAY[21].sErrWTXT:=" 输入的参数mfc9有误";// Error 信息 分配

gErrorARRAY[22].eErrLevel:=Error_Level_4;// Error Level 分配
gErrorARRAY[22].sErrTXT:='Par rfPoint_Power input error.';// Error 信息 分配
gErrorARRAY[22].sErrWTXT:=" 输入的参数rfPoint_Power有误";// Error 信息 分配

gErrorARRAY[23].eErrLevel:=Error_Level_4;// Error Level 分配
gErrorARRAY[23].sErrTXT:='Par par_2 input error.';// Error 信息 分配
gErrorARRAY[23].sErrWTXT:=" 输入的参数par_2有误";// Error 信息 分配

gErrorARRAY[24].eErrLevel:=Error_Level_4;// Error Level 分配
gErrorARRAY[24].sErrTXT:='Par par_3 input error.';// Error 信息 分配
gErrorARRAY[24].sErrWTXT:=" 输入的参数par_3有误";// Error 信息 分配

gErrorARRAY[30].eErrLevel:=Error_Level_3;// Error Level 分配
gErrorARRAY[30].sErrTXT:='Recipe Error (does not exist).';// Error 信息 分配
gErrorARRAY[30].sErrWTXT:=" 配方出错，不存在或配方参数出错.";// Error 信息 分配
//////////////////////////////////////////////////////////////////////////////////////////////////50-500 Machine 

gErrorARRAY[50].eErrLevel:=Error_Level_3;// Error Level 分配
gErrorARRAY[50].sErrTXT:='The air supply conditions are not met: it is not turned on or the air pressure is insufficient.';// Error 信息 分配
gErrorARRAY[50].sErrWTXT:=" 气源条件未满足：未打开或气压不足.";// Error 信息 分配

gErrorARRAY[51].eErrLevel:=Error_Level_3;// Error Level 分配
gErrorARRAY[51].sErrTXT:='The water source conditions are not met: it is not opened or the water flow is insufficient, and the water temperature is overwarm.';// Error 信息 分配
gErrorARRAY[51].sErrWTXT:=" 水源条件未满足：未打开或水流不足、水温超温.";// Error 信息 分配

gErrorARRAY[52].eErrLevel:=Error_Level_3;// Error Level 分配
gErrorARRAY[52].sErrTXT:='Power condition not met: Not powered on or not in a ready state.';// Error 信息 分配
gErrorARRAY[52].sErrWTXT:=" 电源条件未满足：未上电或未进入就绪状态。";// Error 信息 分配

gErrorARRAY[53].eErrLevel:=Error_Level_3;// Error Level 分配
gErrorARRAY[53].sErrTXT:='ForLinGauge Error:disconected or Par. out of limit.';// Error 信息 分配
gErrorARRAY[53].sErrWTXT:=" 前置真空计报错：未链接或读数超限。";// Error 信息 分配

gErrorARRAY[54].eErrLevel:=Error_Level_3;// Error Level 分配
gErrorARRAY[54].sErrTXT:='LoadLockeGauge Error:disconected or Par. out of limit.';// Error 信息 分配
gErrorARRAY[54].sErrWTXT:=" 过渡腔真空计：未链接或读数超限。";// Error 信息 分配

gErrorARRAY[55].eErrLevel:=Error_Level_3;// Error Level 分配
gErrorARRAY[55].sErrTXT:='AIMGauge Error:disconected or Par. out of limit.';// Error 信息 分配
gErrorARRAY[55].sErrWTXT:=" 工艺腔电离真空计：未链接或读数超限。";// Error 信息 分配

gErrorARRAY[56].eErrLevel:=Error_Level_3;// Error Level 分配
gErrorARRAY[56].sErrTXT:='ChamberGauge Error:disconected or Par. out of limit.';// Error 信息 分配
gErrorARRAY[56].sErrWTXT:=" 腔体真空计：未链接或读数超限。";// Error 信息 分配

gErrorARRAY[57].eErrLevel:=Error_Level_3;// Error Level 分配
gErrorARRAY[57].sErrTXT:='Power condition not met: Not powered on or not in a ready state.';// Error 信息 分配
gErrorARRAY[57].sErrWTXT:=" 起破条件不满足，未上电或未就绪。";// Error 信息 分配

gErrorARRAY[58].eErrLevel:=Error_Level_3;// Error Level 分配
gErrorARRAY[58].sErrTXT:='TruboPum tail pressure error or disconected.';// Error 信息 分配
gErrorARRAY[58].sErrWTXT:=" 分子泵尾排压力报错或模块未连接。";// Error 信息 分配

// 100-200 半自动报错
gErrorARRAY[100].eErrLevel:=Error_Level_3;// Error Level 分配
gErrorARRAY[100].sErrTXT:=' CO-Control RF Open Condition Not Satisfied.';// Error 信息 分配
gErrorARRAY[100].sErrWTXT:=" 共同控制RF 起破条件不满足！";// Error 信息 分配

gErrorARRAY[101].eErrLevel:=Error_Level_3;// Error Level 分配
gErrorARRAY[101].sErrTXT:=' CO-Control RF Error.';// Error 信息 分配
gErrorARRAY[101].sErrWTXT:=" 共同控制RF 电源起破过程存在错误！";// Error 信息 分配

gErrorARRAY[102].eErrLevel:=Error_Level_3;// Error Level 分配
gErrorARRAY[102].sErrTXT:=' CO-Control RF Close Condition Not Satisfied.';// Error 信息 分配
gErrorARRAY[102].sErrWTXT:=" 共同控制RF 电源起破过程存在错误！";// Error 信息 分配

gErrorARRAY[103].eErrLevel:=Error_Level_3;// Error Level 分配
gErrorARRAY[103].sErrTXT:=' Open PDV need TB No rotation or open done.';// Error 信息 分配
gErrorARRAY[103].sErrWTXT:=" 开PDV需要分子完全静止或者开启完成才可以操作！";// Error 信息 分配

gErrorARRAY[104].eErrLevel:=Error_Level_3;// Error Level 分配
gErrorARRAY[104].sErrTXT:=' Open PDV sT.:The anterior and posterior differential pressure must be less than 500mTorr';// Error 信息 分配
gErrorARRAY[104].sErrWTXT:=" 开PDV需要前后压差小于500mTorr！";// Error 信息 分配

gErrorARRAY[105].eErrLevel:=Error_Level_3;// Error Level 分配
gErrorARRAY[105].sErrTXT:=' Running State Error';// Error 信息 分配
gErrorARRAY[105].sErrWTXT:=" 运行状态出错！";// Error 信息 分配

gErrorARRAY[106].eErrLevel:=Error_Level_3;// Error Level 分配
gErrorARRAY[106].sErrTXT:=' Actuator Recovery POU Action Time Out';// Error 信息 分配
gErrorARRAY[106].sErrWTXT:=" 执行器复位程序动作超时！";// Error 信息 分配

gErrorARRAY[107].eErrLevel:=Error_Level_3;// Error Level 分配
gErrorARRAY[107].sErrTXT:=' Gauge State Error';// Error 信息 分配
gErrorARRAY[107].sErrWTXT:=" 真空计状态出错！";// Error 信息 分配

gErrorARRAY[108].eErrLevel:=Error_Level_3;// Error Level 分配
gErrorARRAY[108].sErrTXT:=' Chamber Vent POU Action Time Out';// Error 信息 分配
gErrorARRAY[108].sErrWTXT:=" 腔体破空程序动作超时！";// Error 信息 分配

gErrorARRAY[109].eErrLevel:=Error_Level_3;// Error Level 分配
gErrorARRAY[109].sErrTXT:=' LoadLock Vent POU Action Time Out';// Error 信息 分配
gErrorARRAY[109].sErrWTXT:=" LoadLock破空程序动作超时！";// Error 信息 分配

gErrorARRAY[110].eErrLevel:=Error_Level_3;// Error Level 分配
gErrorARRAY[110].sErrTXT:=' Load Wafer POU Action Time Out';// Error 信息 分配
gErrorARRAY[110].sErrWTXT:=" Load Wafer程序动作超时！";// Error 信息 分配

gErrorARRAY[111].eErrLevel:=Error_Level_3;// Error Level 分配
gErrorARRAY[111].sErrTXT:=' ARM IN Action Time Out';// Error 信息 分配
gErrorARRAY[111].sErrWTXT:=" ARM进入腔体动作超时！";// Error 信息 分配

gErrorARRAY[112].eErrLevel:=Error_Level_3;// Error Level 分配
gErrorARRAY[112].sErrTXT:=' Machine Vent POU Time Out';// Error 信息 分配
gErrorARRAY[112].sErrWTXT:=" Machine Vent程序动作超时！";// Error 信息 分配

gErrorARRAY[113].eErrLevel:=Error_Level_3;// Error Level 分配
gErrorARRAY[113].sErrTXT:=' RoughPumpong POU Time Out';// Error 信息 分配
gErrorARRAY[113].sErrWTXT:=" RoughPumpong(粗抽)程序动作超时！";// Error 信息 分配

gErrorARRAY[114].eErrLevel:=Error_Level_3;// Error Level 分配
gErrorARRAY[114].sErrTXT:=' UnLoad Wafer POU Time Out';// Error 信息 分配
gErrorARRAY[114].sErrWTXT:=" UnLoad Wafer程序动作超时！";// Error 信息 分配

gErrorARRAY[115].eErrLevel:=Error_Level_3;// Error Level 分配
gErrorARRAY[115].sErrTXT:=' UnLoad Wafer Arm have wafer,Not allow to UnLoad Wafer';// Error 信息 分配
gErrorARRAY[115].sErrWTXT:=" UnLoad Wafer程序检测到ARM上有晶圆，不允许下晶圆！";// Error 信息 分配

gErrorARRAY[116].eErrLevel:=Error_Level_3;// Error Level 分配
gErrorARRAY[116].sErrTXT:=' Etching POU Run but wafer outside chamber';// Error 信息 分配
gErrorARRAY[116].sErrWTXT:=" 刻蚀程序运行但是腔体内无Wafer！";// Error 信息 分配

gErrorARRAY[120].eErrLevel:=Error_Level_3;// Error Level 分配
gErrorARRAY[120].sErrTXT:=' Gas flow error';// Error 信息 分配
gErrorARRAY[120].sErrWTXT:=" 气体流量出错！";// Error 信息 分配

gErrorARRAY[121].eErrLevel:=Error_Level_3;// Error Level 分配
gErrorARRAY[121].sErrTXT:=' Gas flow not clear';// Error 信息 分配
gErrorARRAY[121].sErrWTXT:=" 气体未关闭，需手动关闭后再执行操作！";// Error 信息 分配

gErrorARRAY[122].eErrLevel:=Error_Level_3;// Error Level 分配
gErrorARRAY[122].sErrTXT:=' LoadLock Pumping TimeOut';// Error 信息 分配
gErrorARRAY[122].sErrWTXT:=" LL腔抽气动作超时！";// Error 信息 分配

gErrorARRAY[123].eErrLevel:=Error_Level_3;// Error Level 分配
gErrorARRAY[123].sErrTXT:=' Pumping limit vacuum timeout';// Error 信息 分配
gErrorARRAY[123].sErrWTXT:=" Etch腔体抽气极限真空超时超时！";// Error 信息 分配

gErrorARRAY[200].eErrLevel:=Error_Level_3;// Error Level 分配
gErrorARRAY[200].sErrTXT:=' Back Of Helium MFC Set Flow Error';// Error 信息 分配
gErrorARRAY[200].sErrWTXT:=" 背氦MFC流量设置参数异常！";// Error 信息 分配

// 300-500 POU出错
gErrorARRAY[300].eErrLevel:=Error_Level_2;// Error Level 分配
gErrorARRAY[300].sErrTXT:='An error occurred in the status check POU.';// Error 信息 分配
gErrorARRAY[300].sErrWTXT:=" 状态检查POU出错。";// Error 信息 分配

//500-1000 电机及真空吸报错

//轴数据分配在500-1499
////////////////////////////////////////////////////////////////////////////////////////////////次要报错


// 报错可按照上面的示例进行扩展


Demo_ACT();

(*
分配气缸报错
*)
METHOD assignARMError_1
VAR_INPUT
	pPoint:POINTER TO ARMModule;
	nBaseErrID:UDINT;
END_VAR
VAR
	n1:UDINT;
END_VAR
(*
pCy^.errorID:=nBaseErrID;

gErrorARRAY[pCy^.errID].eErrLevel:=Error_Level_3;//Error Level 分配
gErrorARRAY[pCy^.errID].sErrTXT:=pCy^.errTXT;//Error 信息 分配
gErrorARRAY[pCy^.errID].sErrWTXT:=pCy^.errWTXT;//Error 信息 分配
*)
pPoint^.errorID:=nBaseErrID;
FOR n1:=1 TO 5 BY 1 DO
	gErrorARRAY[pPoint^.getErrID(n1)].eErrLevel:=Error_Level_3;//Error Level 分配
	gErrorARRAY[pPoint^.getErrID(n1)].sErrTXT:=pPoint^.getErrTXT(n1);//Error 信息 分配
	gErrorARRAY[pPoint^.getErrID(n1)].sErrWTXT:=pPoint^.getErrWTXT(n1);//Error 信息 分配
END_FOR

IF nInit_ARM<nMaxNum_ARM THEN
	nInit_ARM:=nInit_ARM+1;//计数
	pARMArr[nInit_ARM]:=pPoint;
END_IF
END_METHOD

(*
分配电机报错
*)
METHOD assignAxisError
VAR_INPUT
	pMotor:POINTER TO FB_MotorMovements;
END_VAR
gErrorARRAY[pMotor^.stMotorOutput.axisErrId].eErrLevel:=Error_Level_3;//Error Level 分配 
gErrorARRAY[pMotor^.stMotorOutput.axisErrId].sErrTXT:=pMotor^.stMotorOutput.axisErrTxt;//Error 信息 分配
gErrorARRAY[pMotor^.stMotorOutput.axisErrId].sErrWTXT:=pMotor^.stMotorOutput.axisErrWTxt;//Error 信息 分配

IF nInit_Axis<nMaxNum_Axis THEN
	nInit_Axis:=nInit_Axis+1;//计数
	pAxisArr[nInit_Axis]:=pMotor;
END_IF
END_METHOD

(*
分配电机报错
*)
METHOD assignAxisError_1
VAR_INPUT
	pMotor:POINTER TO FB_MotorMovements;
	nBaseErrID:UDINT;
END_VAR
VAR
	n1:UDINT;
END_VAR
(*
pMotor^.nBaseErrID:=nBaseErrID;

gErrorARRAY[pMotor^.stMotorOutput.axisErrId].eErrLevel:=Error_Level_3;//Error Level 分配 
gErrorARRAY[pMotor^.stMotorOutput.axisErrId].sErrTXT:=pMotor^.stMotorOutput.axisErrTxt;//Error 信息 分配
gErrorARRAY[pMotor^.stMotorOutput.axisErrId].sErrWTXT:=pMotor^.stMotorOutput.axisErrWTxt;//Error 信息 分配
*)
pMotor^.nBaseErrID:=nBaseErrID;
pMotor^.stMotorOutput.pMotionModule^.errorID:=nBaseErrID;

FOR n1:=1 TO 16 BY 1 DO
	gErrorARRAY[pMotor^.stMotorOutput.pMotionModule^.getErrID(n1)].eErrLevel:=Error_Level_3;//Error Level 分配 
	gErrorARRAY[pMotor^.stMotorOutput.pMotionModule^.getErrID(n1)].sErrTXT:=pMotor^.stMotorOutput.pMotionModule^.getErrTXT(n1);//Error 信息 分配
	gErrorARRAY[pMotor^.stMotorOutput.pMotionModule^.getErrID(n1)].sErrWTXT:=pMotor^.stMotorOutput.pMotionModule^.getErrWTXT(n1);//Error 信息 分配
END_FOR


IF nInit_Axis<nMaxNum_Axis THEN
	nInit_Axis:=nInit_Axis+1;//计数
	pAxisArr[nInit_Axis]:=pMotor;
END_IF
END_METHOD

(*
分配气缸报错
*)
METHOD assignChillerError_1
VAR_INPUT
	pPoint:POINTER TO ChillerModule_1;
	nBaseErrID:UDINT;
END_VAR
VAR
	n1:UDINT;
END_VAR
(*
pCy^.errorID:=nBaseErrID;

gErrorARRAY[pCy^.errID].eErrLevel:=Error_Level_3;//Error Level 分配
gErrorARRAY[pCy^.errID].sErrTXT:=pCy^.errTXT;//Error 信息 分配
gErrorARRAY[pCy^.errID].sErrWTXT:=pCy^.errWTXT;//Error 信息 分配
*)
pPoint^.errorID:=nBaseErrID;
FOR n1:=1 TO 4 BY 1 DO
	gErrorARRAY[pPoint^.getErrID(n1)].eErrLevel:=Error_Level_3;//Error Level 分配
	gErrorARRAY[pPoint^.getErrID(n1)].sErrTXT:=pPoint^.getErrTXT(n1);//Error 信息 分配
	gErrorARRAY[pPoint^.getErrID(n1)].sErrWTXT:=pPoint^.getErrWTXT(n1);//Error 信息 分配
END_FOR

IF nInit_Chiller<nMaxNum_Chiller THEN
	nInit_Chiller:=nInit_Chiller+1;//计数
	pChillerArr[nInit_Chiller]:=pPoint;
END_IF
END_METHOD

(*
分配气缸报错
*)
METHOD assignCyError
VAR_INPUT
	pCy:POINTER TO CylinderModule;
END_VAR
gErrorARRAY[pCy^.errID].eErrLevel:=Error_Level_3;//Error Level 分配
gErrorARRAY[pCy^.errID].sErrTXT:=pCy^.errTXT;//Error 信息 分配
gErrorARRAY[pCy^.errID].sErrWTXT:=pCy^.errWTXT;//Error 信息 分配

IF nInit_Cy<nMaxNum_Cy THEN
	nInit_Cy:=nInit_Cy+1;//计数
	pCyArr[nInit_Cy]:=pCy;
END_IF
END_METHOD

(*
分配气缸报错
*)
METHOD assignCyError_1
VAR_INPUT
	pCy:POINTER TO CylinderModule;
	nBaseErrID:UDINT;
END_VAR
VAR
	n1:UDINT;
END_VAR
(*
pCy^.errorID:=nBaseErrID;

gErrorARRAY[pCy^.errID].eErrLevel:=Error_Level_3;//Error Level 分配
gErrorARRAY[pCy^.errID].sErrTXT:=pCy^.errTXT;//Error 信息 分配
gErrorARRAY[pCy^.errID].sErrWTXT:=pCy^.errWTXT;//Error 信息 分配
*)
pCy^.errorID:=nBaseErrID;
FOR n1:=1 TO 16 BY 1 DO
	gErrorARRAY[pCy^.getErrID(n1)].eErrLevel:=Error_Level_3;//Error Level 分配
	gErrorARRAY[pCy^.getErrID(n1)].sErrTXT:=pCy^.getErrTXT(n1);//Error 信息 分配
	gErrorARRAY[pCy^.getErrID(n1)].sErrWTXT:=pCy^.getErrWTXT(n1);//Error 信息 分配
END_FOR

IF nInit_Cy<nMaxNum_Cy THEN
	nInit_Cy:=nInit_Cy+1;//计数
	pCyArr[nInit_Cy]:=pCy;
END_IF
END_METHOD

(*
分配气缸报错
*)
METHOD assignMFCError
VAR_INPUT
	pMFC:POINTER TO MFCModule;
	nBaseErrID:UDINT;
END_VAR
VAR
	n1:UDINT;
END_VAR
(*
pCy^.errorID:=nBaseErrID;

gErrorARRAY[pCy^.errID].eErrLevel:=Error_Level_3;//Error Level 分配
gErrorARRAY[pCy^.errID].sErrTXT:=pCy^.errTXT;//Error 信息 分配
gErrorARRAY[pCy^.errID].sErrWTXT:=pCy^.errWTXT;//Error 信息 分配
*)
pMFC^.errorID:=nBaseErrID;
FOR n1:=1 TO 5 BY 1 DO
	gErrorARRAY[pMFC^.getErrID(n1)].eErrLevel:=Error_Level_3;//Error Level 分配
	gErrorARRAY[pMFC^.getErrID(n1)].sErrTXT:=pMFC^.getErrTXT(n1);//Error 信息 分配
	gErrorARRAY[pMFC^.getErrID(n1)].sErrWTXT:=pMFC^.getErrWTXT(n1);//Error 信息 分配
END_FOR

IF nInit_MFC<nMaxNum_MFC THEN
	nInit_MFC:=nInit_MFC+1;//计数
	pMFCArr[nInit_MFC]:=pMFC;
END_IF
END_METHOD

(*
PDV报错
*)
METHOD assignPDVError_1
VAR_INPUT
	pPoint:POINTER TO PVModule;
	nBaseErrID:UDINT;
END_VAR
VAR
	n1:UDINT;
END_VAR
(*
pCy^.errorID:=nBaseErrID;

gErrorARRAY[pCy^.errID].eErrLevel:=Error_Level_3;//Error Level 分配
gErrorARRAY[pCy^.errID].sErrTXT:=pCy^.errTXT;//Error 信息 分配
gErrorARRAY[pCy^.errID].sErrWTXT:=pCy^.errWTXT;//Error 信息 分配
*)
pPoint^.errorID:=nBaseErrID;
FOR n1:=1 TO 5 BY 1 DO
	gErrorARRAY[pPoint^.getErrID(n1)].eErrLevel:=Error_Level_3;//Error Level 分配
	gErrorARRAY[pPoint^.getErrID(n1)].sErrTXT:=pPoint^.getErrTXT(n1);//Error 信息 分配
	gErrorARRAY[pPoint^.getErrID(n1)].sErrWTXT:=pPoint^.getErrWTXT(n1);//Error 信息 分配
END_FOR

IF nInit_PDV<nMaxNum_PDV THEN
	nInit_PDV:=nInit_PDV+1;//计数
	pPDVArr[nInit_PDV]:=pPoint;
END_IF
END_METHOD

(*
分配气缸报错
*)
METHOD assignRFError_1
VAR_INPUT
	pPoint:POINTER TO RFModule;
	nBaseErrID:UDINT;
END_VAR
VAR
	n1:UDINT;
END_VAR
(*
pCy^.errorID:=nBaseErrID;

gErrorARRAY[pCy^.errID].eErrLevel:=Error_Level_3;//Error Level 分配
gErrorARRAY[pCy^.errID].sErrTXT:=pCy^.errTXT;//Error 信息 分配
gErrorARRAY[pCy^.errID].sErrWTXT:=pCy^.errWTXT;//Error 信息 分配
*)
pPoint^.errorID:=nBaseErrID;
FOR n1:=1 TO 6 BY 1 DO
	gErrorARRAY[pPoint^.getErrID(n1)].eErrLevel:=Error_Level_3;//Error Level 分配
	gErrorARRAY[pPoint^.getErrID(n1)].sErrTXT:=pPoint^.getErrTXT(n1);//Error 信息 分配
	gErrorARRAY[pPoint^.getErrID(n1)].sErrWTXT:=pPoint^.getErrWTXT(n1);//Error 信息 分配
END_FOR

IF nInit_RF<nMaxNum_RF THEN
	nInit_RF:=nInit_RF+1;//计数
	pRFArr[nInit_RF]:=pPoint;
END_IF
END_METHOD

(*
分配气缸报错
*)
METHOD assignRFError_2
VAR_INPUT
	pPoint:POINTER TO RFModule_Source;
	nBaseErrID:UDINT;
END_VAR
VAR
	n1:UDINT;
END_VAR
(*
pCy^.errorID:=nBaseErrID;

gErrorARRAY[pCy^.errID].eErrLevel:=Error_Level_3;//Error Level 分配
gErrorARRAY[pCy^.errID].sErrTXT:=pCy^.errTXT;//Error 信息 分配
gErrorARRAY[pCy^.errID].sErrWTXT:=pCy^.errWTXT;//Error 信息 分配
*)
pPoint^.errorID:=nBaseErrID;
FOR n1:=1 TO 6 BY 1 DO
	gErrorARRAY[pPoint^.getErrID(n1)].eErrLevel:=Error_Level_3;//Error Level 分配
	gErrorARRAY[pPoint^.getErrID(n1)].sErrTXT:=pPoint^.getErrTXT(n1);//Error 信息 分配
	gErrorARRAY[pPoint^.getErrID(n1)].sErrWTXT:=pPoint^.getErrWTXT(n1);//Error 信息 分配
END_FOR

IF nInit_RF<nMaxNum_RF THEN
	nInit_RF:=nInit_RF+1;//计数
	pRFArr[nInit_RF]:=pPoint;
END_IF
END_METHOD

(*
分配气缸报错
*)
METHOD assignTMPError_1
VAR_INPUT
	pPoint:POINTER TO TMPModule;
	nBaseErrID:UDINT;
END_VAR
VAR
	n1:UDINT;
END_VAR
(*
pCy^.errorID:=nBaseErrID;

gErrorARRAY[pCy^.errID].eErrLevel:=Error_Level_3;//Error Level 分配
gErrorARRAY[pCy^.errID].sErrTXT:=pCy^.errTXT;//Error 信息 分配
gErrorARRAY[pCy^.errID].sErrWTXT:=pCy^.errWTXT;//Error 信息 分配
*)
pPoint^.errorID:=nBaseErrID;
FOR n1:=1 TO 6 BY 1 DO
	gErrorARRAY[pPoint^.getErrID(n1)].eErrLevel:=Error_Level_3;//Error Level 分配
	gErrorARRAY[pPoint^.getErrID(n1)].sErrTXT:=pPoint^.getErrTXT(n1);//Error 信息 分配
	gErrorARRAY[pPoint^.getErrID(n1)].sErrWTXT:=pPoint^.getErrWTXT(n1);//Error 信息 分配
END_FOR

IF nInit_TMP<nMaxNum_TMP THEN
	nInit_TMP:=nInit_TMP+1;//计数
	pTMPArr[nInit_TMP]:=pPoint;
END_IF
END_METHOD

(*
分配气缸报错
*)
METHOD assignVPEError_1
VAR_INPUT
	pPoint:POINTER TO VPEModule;
	nBaseErrID:UDINT;
END_VAR
VAR
	n1:UDINT;
END_VAR
(*
pCy^.errorID:=nBaseErrID;

gErrorARRAY[pCy^.errID].eErrLevel:=Error_Level_3;//Error Level 分配
gErrorARRAY[pCy^.errID].sErrTXT:=pCy^.errTXT;//Error 信息 分配
gErrorARRAY[pCy^.errID].sErrWTXT:=pCy^.errWTXT;//Error 信息 分配
*)
pPoint^.errorID:=nBaseErrID;
FOR n1:=1 TO 8 BY 1 DO
	gErrorARRAY[pPoint^.getErrID(n1)].eErrLevel:=Error_Level_3;//Error Level 分配
	gErrorARRAY[pPoint^.getErrID(n1)].sErrTXT:=pPoint^.getErrTXT(n1);//Error 信息 分配
	gErrorARRAY[pPoint^.getErrID(n1)].sErrWTXT:=pPoint^.getErrWTXT(n1);//Error 信息 分配
END_FOR

IF nInit_Vpe<nMaxNum_Vpe THEN
	nInit_Vpe:=nInit_Vpe+1;//计数
	pVpeArr[nInit_Vpe]:=pPoint;
END_IF
END_METHOD

ACTION Demo_ACT:
// 电机
IF NOT bInit_Axis THEN
	nInit_Axis:=0;
	// bInit_Axis:=TRUE;
	
	// 电机：(500~1499)
//	assignAxisError_1(ADR(gLoad_AXIS.CY1Axis),500);
//	assignAxisError_1(ADR(gUnLoad_AXIS.CY1Axis),520);
//	assignAxisError_1(ADR(gLoad_AXIS.X1Axis),540);
//	assignAxisError_1(ADR(gLoad_AXIS.Y1Axis),560);
//	assignAxisError_1(ADR(gLoad_AXIS.Z1Axis),580);
//	assignAxisError_1(ADR(gLoad_AXIS.R1Axis),600);
	
//	assignAxisError_1(ADR(gTestSocket_AXIS.X1AXIS),700);
//	assignAxisError_1(ADR(gTestSocket_AXIS.Z1AXIS),720);
//	assignAxisError_1(ADR(gTestSocket_AXIS.R1AXIS),740);
//	assignAxisError_1(ADR(gTestSocket_AXIS.Y1AXIS),760);
//	assignAxisError_1(ADR(gTestSocket_AXIS.UX2AXIS),780);
//	assignAxisError_1(ADR(gTestSocket_AXIS.UY2AXIS),800);
//	assignAxisError_1(ADR(gTestSocket_AXIS.X3AXIS),820);

//	assignAxisError_1(ADR(gCoaxial_AXIS.Y1AXIS),900);
	
	
//	assignAxisError_1(ADR(gRXTest_AXIS.Z1AXIS),1000);
//	assignAxisError_1(ADR(gRXTest_AXIS.X1AXIS),1020);
//	assignAxisError_1(ADR(gRXTest_AXIS.Y1AXIS),1040);
//	assignAxisError_1(ADR(gRXTest_AXIS.U1AXIS),1060);
//	assignAxisError_1(ADR(gRXTest_AXIS.Y2AXIS),1080);
//	assignAxisError_1(ADR(gRXTest_AXIS.CZ2AXIS),1100);
//	assignAxisError_1(ADR(gRXTest_AXIS.CZ3AXIS),1120);
//	assignAxisError_1(ADR(gRXTest_AXIS.CY3AXIS),1140);
	
//	assignAxisError_1(ADR(gTXTest_AXIS.Y1AXIS),1200);
	
//	assignAxisError_1(ADR(gUnLoad_AXIS.X1Axis),1300);
//	assignAxisError_1(ADR(gUnLoad_AXIS.Y1Axis),1320);
//	assignAxisError_1(ADR(gUnLoad_AXIS.Z1Axis),1340);
//	assignAxisError_1(ADR(gUnLoad_AXIS.R1Axis),1360);
//	assignAxisError_1(ADR(gUnLoad_AXIS.X2Axis),1380);
	
END_IF
// TMP
// 分子泵，根据腔体总数量决定，每个腔体至少百分之60在工作；
IF NOT bInit_TMP THEN
	nInit_TMP:=0;
	assignTMPError_1(ADR(gICP.TruboPum),2500);
END_IF
// PDV
IF NOT bInit_PDV THEN
	nInit_PDV:=0;
	assignPDVError_1(ADR(gICP.PDV),2720);
END_IF

// 气缸
IF NOT bInit_Cy THEN
	nInit_Cy:=0;
	assignCyError_1(ADR(gICP.ForlinLineValve),2010);
	assignCyError_1(ADR(gICP.RoughValve),2020);
	assignCyError_1(ADR(gICP.SlowPummingValve),2030);
	assignCyError_1(ADR(gICP.FastPummingValve),2040);
	assignCyError_1(ADR(gICP.ElectrodeCyl),2050);
	assignCyError_1(ADR(gICP.LiftPinCyl),2060);
	
	assignCyError_1(ADR(gICP.GVA1Valve),2070);
	assignCyError_1(ADR(gICP.GVA2Valve),2080);
	assignCyError_1(ADR(gICP.GVA3Valve),2090);
	assignCyError_1(ADR(gICP.GVA4Valve),2100);
	assignCyError_1(ADR(gICP.GVA5Valve),2110);
	assignCyError_1(ADR(gICP.GVA6Valve),2120);
	assignCyError_1(ADR(gICP.GVA7Valve),2130);
	assignCyError_1(ADR(gICP.GVA8Valve),2140);
	assignCyError_1(ADR(gICP.GVA9Valve),2260);
	assignCyError_1(ADR(gICP.GVA10Valve_Vent),2270);
	assignCyError_1(ADR(gICP.GV20Valve_Main),2340);
	
	assignCyError_1(ADR(gICP.GVB1Valve),2150);
	assignCyError_1(ADR(gICP.GVB2Valve),2160);
	assignCyError_1(ADR(gICP.GVB3Valve),2170);
	assignCyError_1(ADR(gICP.GVB4Valve),2180);
	assignCyError_1(ADR(gICP.GVB5Valve),2190);
	assignCyError_1(ADR(gICP.GVB6Valve),2200);
	assignCyError_1(ADR(gICP.GVB7Valve),2210);
	assignCyError_1(ADR(gICP.GVB8Valve),2280);
	assignCyError_1(ADR(gICP.GVB9Valve),2290);
	
	assignCyError_1(ADR(gICP.ISOValve),2220);
	assignCyError_1(ADR(gICP.AIMValve),2230);
	assignCyError_1(ADR(gICP.GateDoorValve),2240);
	assignCyError_1(ADR(gICP.VentValve),2250);
	assignCyError_1(ADR(gICP.GASBoxVentValve),2300);
	assignCyError_1(ADR(gICP.HeINValve),2310);
	assignCyError_1(ADR(gICP.HePumValve),2320);
	assignCyError_1(ADR(gICP.TBPurgeValve),2350);
END_IF

IF NOT bInit_MFC THEN
	nInit_MFC:=0;
	assignMFCError(ADR(gICP.MFC1),2600);
	assignMFCError(ADR(gICP.MFC2),2610);
	assignMFCError(ADR(gICP.MFC3),2620);
	assignMFCError(ADR(gICP.MFC4),2630);
	assignMFCError(ADR(gICP.MFC5),2640);
	assignMFCError(ADR(gICP.MFC6),2650);
	assignMFCError(ADR(gICP.MFC7),2660);
END_IF
IF NOT bInit_RF THEN
	nInit_RF:=0;
	assignRFError_1(ADR(gICP.PowerRF),2700);
	assignRFError_2(ADR(gICP.SourceRF),2710);
END_IF

IF NOT bInit_Chiller THEN
	nInit_Chiller:=0;
	assignChillerError_1(ADR(gICP.Chiller),2800);
END_IF

IF NOT bInit_ARM THEN
	nInit_ARM:=0;
	assignARMError_1(ADR(gICP.ARM),2330);
END_IF


// 电机报警监控
FOR nTemp_Axis:=1 TO nInit_Axis BY 1 DO
	r_trig_AxisArr[nTemp_Axis](CLK:=(pAxisArr[nTemp_Axis]^.Get_Error()) AND (''<>pAxisArr[nTemp_Axis]^.Get_ErrTxt()));
	IF r_trig_AxisArr[nTemp_Axis].Q THEN
		error_Trigger(TO_DINT(pAxisArr[nTemp_Axis]^.Get_ErrID()));
	END_IF
END_FOR
//电磁阀报警监控
FOR nTemp_Cy:=1 TO nInit_Cy BY 1 DO
	r_trig_CyArr[nTemp_Cy](CLK:=(pCyArr[nTemp_Cy]^.error) AND (''<>pCyArr[nTemp_Cy]^.errTXT));
	IF r_trig_CyArr[nTemp_Cy].Q THEN
		IF pCyArr[nTemp_Cy]^.cylinderType<>CylinderType.CylinderType_Vacuum THEN
			error_Trigger(TO_DINT(pCyArr[nTemp_Cy]^.errID));
		END_IF
	END_IF
END_FOR

//MFC
FOR nTemp_MFC:=1 TO nInit_MFC BY 1 DO
	r_trig_MFCArr[nTemp_MFC](CLK:=(pMFCArr[nTemp_MFC]^.error) AND (''<>pMFCArr[nTemp_MFC]^.errTXT));
	IF r_trig_MFCArr[nTemp_MFC].Q THEN
		error_Trigger(TO_DINT(pMFCArr[nTemp_MFC]^.errID));
	END_IF
END_FOR

//VPE
FOR nTemp_Vpe:=1 TO nInit_Vpe BY 1 DO
	r_trig_VpeArr[nTemp_Vpe](CLK:=(pVpeArr[nTemp_Vpe]^.error) AND (''<>pVpeArr[nTemp_Vpe]^.errTXT));
	IF r_trig_VpeArr[nTemp_Vpe].Q THEN
		error_Trigger(TO_DINT(pVpeArr[nTemp_Vpe]^.errID));
	END_IF
END_FOR
//TMP
FOR nTemp_TMP:=1 TO nInit_TMP BY 1 DO
	r_trig_TMPArr[nTemp_TMP](CLK:=(pTMPArr[nTemp_TMP]^.error) AND (''<>pTMPArr[nTemp_TMP]^.errTXT));
	IF r_trig_TMPArr[nTemp_TMP].Q THEN
		error_Trigger(TO_DINT(pTMPArr[nTemp_TMP]^.errID));
	END_IF
END_FOR
//PDV
FOR nTemp_PDV:=1 TO nInit_PDV BY 1 DO
	r_trig_PDVArr[nTemp_PDV](CLK:=(pPDVArr[nTemp_PDV]^.error) AND (''<>pPDVArr[nTemp_PDV]^.errTXT));
	IF r_trig_PDVArr[nTemp_PDV].Q THEN
		error_Trigger(TO_DINT(pPDVArr[nTemp_PDV]^.errID));
	END_IF
END_FOR
//RF
FOR nTemp_RF:=1 TO nInit_RF BY 1 DO
	r_trig_RFArr[nTemp_RF](CLK:=(pRFArr[nTemp_RF]^.error) AND (''<>pRFArr[nTemp_RF]^.errTXT));
	IF r_trig_RFArr[nTemp_RF].Q THEN
		error_Trigger(TO_DINT(pRFArr[nTemp_RF]^.errID));
	END_IF
END_FOR

//Chiller
FOR nTemp_Chiller:=1 TO nInit_Chiller BY 1 DO
	r_trig_ChillerArr[nTemp_Chiller](CLK:=(pChillerArr[nTemp_Chiller]^.error) AND (''<>pChillerArr[nTemp_Chiller]^.errTXT));
	IF r_trig_ChillerArr[nTemp_Chiller].Q THEN
		error_Trigger(TO_DINT(pChillerArr[nTemp_Chiller]^.errID));
	END_IF
END_FOR

//ARM
FOR nTemp_ARM:=1 TO nInit_ARM BY 1 DO
	r_trig_ARMArr[nTemp_ARM](CLK:=(pARMArr[nTemp_ARM]^.error) AND (''<>pARMArr[nTemp_ARM]^.errTXT));
	IF r_trig_ARMArr[nTemp_ARM].Q THEN
		error_Trigger(TO_DINT(pARMArr[nTemp_ARM]^.errID));
	END_IF
END_FOR
END_ACTION

METHOD PRIVATE Demo_Reset : BOOL
VAR_INPUT
END_VAR
VAR
	LRobot_Index_reset:INT;
	Test_Index_reset:INT;
	Buff_Index_reset:INT;
	BIN1_Index_reset:INT;
	BIN2_Index_reset:INT;
	ULRobot_Index_reset:INT;
	i: INT;
END_VAR

//(***********  ***********)

// Valve
gICP.ForlinLineValve.Act_Reset();	
gICP.RoughValve.Act_Reset();
gICP.SlowPummingValve.Act_Reset();
gICP.FastPummingValve.Act_Reset();
gICP.ElectrodeCyl.Act_Reset();
gICP.LiftPinCyl.Act_Reset();

gICP.GVA1Valve.Act_Reset();
gICP.GVA2Valve.Act_Reset();
gICP.GVA3Valve.Act_Reset();
gICP.GVA4Valve.Act_Reset();
gICP.GVA5Valve.Act_Reset();
gICP.GVA6Valve.Act_Reset();
gICP.GVA7Valve.Act_Reset();
gICP.GVA8Valve.Act_Reset();
gICP.GVA9Valve.Act_Reset();
gICP.GVA10Valve_Vent.Act_Reset();

gICP.GVB1Valve.Act_Reset();
gICP.GVB2Valve.Act_Reset();
gICP.GVB3Valve.Act_Reset();
gICP.GVB4Valve.Act_Reset();
gICP.GVB5Valve.Act_Reset();
gICP.GVB6Valve.Act_Reset();
gICP.GVB7Valve.Act_Reset();
gICP.GVB8Valve.Act_Reset();
gICP.GVB9Valve.Act_Reset();
gICP.GV20Valve_Main.Act_Reset();


gICP.ISOValve.Act_Reset();
gICP.AIMValve.Act_Reset();
gICP.GateDoorValve.Act_Reset();
gICP.VentValve.Act_Reset();

gICP.TBPurgeValve.Act_Reset();
gICP.HeINValve.Act_Reset();
gICP.HePumValve.Act_Reset();

// MFC 
gICP.MFC1.Act_Reset();	
gICP.MFC2.Act_Reset();
gICP.MFC3.Act_Reset();
gICP.MFC4.Act_Reset();
gICP.MFC5.Act_Reset();
gICP.MFC6.Act_Reset();
gICP.MFC7.Act_Reset();
// TB
gICP.TruboPum.Act_Reset();	
// PDV 
gICP.PDV.Act_Reset();
// RF 
gICP.SourceRF.Act_Reset();
gICP.PowerRF.Act_Reset();
// Chiller
gICP.Chiller.Act_Reset();
// Chiller
gICP.ARM.Act_Reset();
END_METHOD

METHOD getErrTXT : STRING(255)
VAR_INPUT
	errorID					:DINT;
END_VAR
VAR
	sErrTXT					:STRING(255);
END_VAR
sErrTXT:='';
sErrTXT:=CONCAT(sErrTXT,CONCAT('ID:',TO_STRING(gErrorARRAY[errorID].uErrID)));
sErrTXT:=CONCAT(sErrTXT,',');
sErrTXT:=CONCAT(sErrTXT,CONCAT('Level:',TO_STRING(gErrorARRAY[errorID].eErrLevel)));
sErrTXT:=CONCAT(sErrTXT,',');
sErrTXT:=CONCAT(sErrTXT,CONCAT('ErrMsg:',gErrorARRAY[errorID].sErrTXT));
getErrTXT:=sErrTXT;
END_METHOD

METHOD getErrWTXT : WSTRING(255)
VAR_INPUT
	errorID					:DINT;
END_VAR
VAR
	sErrTXT					:WSTRING(255);
END_VAR
sErrTXT:="";
sErrTXT:=WCONCAT(sErrTXT,WCONCAT("ID：",TO_WSTRING(gErrorARRAY[errorID].uErrID)));
sErrTXT:=WCONCAT(sErrTXT,"，");
sErrTXT:=WCONCAT(sErrTXT,WCONCAT("等级：",TO_WSTRING(gErrorARRAY[errorID].eErrLevel)));
sErrTXT:=WCONCAT(sErrTXT,"，");
sErrTXT:=WCONCAT(sErrTXT,WCONCAT("错误信息：",gErrorARRAY[errorID].sErrWTXT));
getErrWTXT:=sErrTXT;
END_METHOD

//触发各个通讯对象复位
METHOD resetFunc : BOOL
VAR_INPUT
END_VAR
VAR
	iTempReset:DINT:=0;
	indexArr_temp_reset:ARRAY [0..g_Max_Data_Elements] OF DINT;
	index_temp_reset:DINT;
	index_temp_reset_remove:DINT;
END_VAR
(*********** DOE ***********)
	Demo_Reset();

(*********** 公共部分 ***********)
	FOR iTempReset:=g_d_ErrorBegin TO g_d_ErrorEnd DO
		gErrorARRAY[iTempReset].bError:=FALSE;
	END_FOR
	
	index_temp_reset:=0;
	gError_fbTable.A_GetFirst(putPosPtr:=0,hTable:=gError_hTable);
	IF gError_fbTable.bOk THEN
		//gError_fbTable.A_Remove(key:=gError_fbTable.getPosPtr,hTable:=gError_hTable);
		//gError_fbTable.A_Remove(key:=gError_fbTable.getValue,hTable:=gError_hTable);
		indexArr_temp_reset[index_temp_reset]:=TO_DINT(gError_fbTable.getValue);
		REPEAT
			gError_fbTable.A_GetNext(putPosPtr:=gError_fbTable.getPosPtr,hTable:=gError_hTable);
			IF gError_fbTable.bOk THEN
				index_temp_reset:=index_temp_reset+1;
				indexArr_temp_reset[index_temp_reset]:=TO_DINT(gError_fbTable.getValue);
			END_IF
		UNTIL NOT gError_fbTable.bOk
		END_REPEAT
	END_IF
	FOR index_temp_reset_remove:=0 TO index_temp_reset BY 1 DO
		gError_fbTable.A_Remove(key:=TO_WORD(indexArr_temp_reset[index_temp_reset_remove]),hTable:=gError_hTable);
	END_FOR
END_METHOD

//触发各个通讯对象复位
METHOD resetFunc_1 : BOOL
VAR_INPUT
END_VAR
VAR
	iTempReset:DINT:=0;
	indexArr_temp_reset:ARRAY [0..g_Max_Data_Elements] OF DINT;
	index_temp_reset:DINT;
	index_temp_reset_remove:DINT;
END_VAR



(*********** 公共部分 ***********)
	FOR iTempReset:=g_d_ErrorBegin TO g_d_ErrorEnd DO
		gErrorARRAY[iTempReset].bError:=FALSE;
	END_FOR
	
	index_temp_reset:=0;
	gError_fbTable.A_GetFirst(putPosPtr:=0,hTable:=gError_hTable);
	IF gError_fbTable.bOk THEN
		//gError_fbTable.A_Remove(key:=gError_fbTable.getPosPtr,hTable:=gError_hTable);
		//gError_fbTable.A_Remove(key:=gError_fbTable.getValue,hTable:=gError_hTable);
		indexArr_temp_reset[index_temp_reset]:=TO_DINT(gError_fbTable.getValue);
		REPEAT
			gError_fbTable.A_GetNext(putPosPtr:=gError_fbTable.getPosPtr,hTable:=gError_hTable);
			IF gError_fbTable.bOk THEN
				index_temp_reset:=index_temp_reset+1;
				indexArr_temp_reset[index_temp_reset]:=TO_DINT(gError_fbTable.getValue);
			END_IF
		UNTIL NOT gError_fbTable.bOk
		END_REPEAT
	END_IF
	FOR index_temp_reset_remove:=0 TO index_temp_reset BY 1 DO
		gError_fbTable.A_Remove(key:=TO_WORD(indexArr_temp_reset[index_temp_reset_remove]),hTable:=gError_hTable);
	END_FOR
END_METHOD

END_PROGRAM

// ---- POUs/BaseModule/ActionModule/motorModule/FB_MotorMovements.TcPOU
FUNCTION_BLOCK FB_MotorMovements
VAR_IN_OUT
	axis							:AXIS_REF;//链接到实际的轴
	WarmHMI							:WARMStruct;
END_VAR
VAR_INPUT
	bPLimitSwitch					:BOOL:=TRUE;//MC轴正限位感应信号
	bNLimitSwitch					:BOOL:=TRUE;//MC轴负限位感应信号
	bDOGPointSwitch					:BOOL:=FALSE;//MC轴原点感应信号
	bTorqueEN						:BOOL:=FALSE;// 启用条件
	bTorqueAlmValue					:LREAL;// 报警扭力值
	bP_Pos							:LREAL:=0.777;	 //正向位置(开门）
	bN_Pos							:LREAL:=0.777;	 //负向位置(关门）

	eMotorType						:MotorType:=MotorType.MotorType_Default;//设置电机的类型
	bModuloMode						:BOOL:=FALSE;// modulo Mode, 旋转模式
	nBaseErrID						:UDINT:=0;//电机错误报警分配的起始ID
	sNameTXT						:STRING(255):='';//电机名字

	bE_Stop							:BOOL:=TRUE;//急停信号
	//eCtrlMode						:ControlMode:=ControlMode.eManualCtrMode;//eManualCtrMode or eAutoCtrMode
	hmiEN							:BOOL:=TRUE;//HMI 启用条件
	
//POWER
	//bPowerEnable					:BOOL:=TRUE;//轴使能触发
	bEnablePositive					:BOOL:=TRUE;//轴允许正转
	bEnableNegative					:BOOL:=TRUE;//轴允许反转
//Soft limit
	bEnableSoftLimit				:BOOL:=FALSE;//轴软限位 启用信号
	fSoftPLimitPos					:LREAL:=9999999;//轴软限位 正向软限位
	fSoftNLimitPos					:LREAL:=-9999999;//轴软限位 负向软限位
	
	bJogConditionOuter				:BOOL:=TRUE;//轴JOG运动启停条件Outer
	bAbsConditionOuter				:BOOL:=TRUE;//轴绝对运动启停条件Outer
	bRelConditionOuter				:BOOL:=TRUE;//轴相对运动启停条件Outer
	bVelConditionOuter				:BOOL:=TRUE;//轴速度模式启停条件Outer
	bSetConditionOuter				:BOOL:=TRUE;//轴当前位置设定启停条件Outer
	bHomeConditionOuter				:BOOL:=TRUE;//轴go home的启停条件Outer
	bMoveModuloConditionOuter		:BOOL:=TRUE;//轴模运动启停条件Outer
	
	bHomeDirection					:BOOL:=TRUE;//轴go home方向 TRUE--正方向，FALSE--负方向
	eHomeMode						:MotorHomeMode:=MotorHomeMode.MotorHomeMode_Default;//轴go home 模式
	fHomeLimitSwitch_To_DOGDistance	:LREAL:=5;//电机Home模式为 MotorHomeMode_PLimitSwitch_To_DOG/MotorHomeMode_NLimitSwitch_To_DOG 时, 脱离限位为原点的距离值
	fHomeOnlyDOGDistance			:LREAL:=5;//电机Home模式为 MotorHomeMode_OnlyDOGPointSwitch 时, 执行往复搜寻动作的幅度
	fHomeOnlyDOGMaxDistance			:LREAL:=360;//电机Home模式为 MotorHomeMode_OnlyDOGPointSwitch 时, 执行往复搜寻动作幅度的最大值
	fHomePosition					:LREAL:=0;
	fHomeCheckRange					:LREAL:=0.01;//轴go home执行完后当前位置判断值
	fHomeVel						:LREAL:=10;//轴go home 查找限位的速率
	fHomeVelSlow					:LREAL:=5;//轴go home 查找限位的爬行速率
	fPosDeviation					:LREAL:=0.01;
	fSoftLimitVel					:LREAL:=5.0;// 速度限制	
	noteWTXT						:WSTRING(255):="";//气缸动作NoteTXT 中文
END_VAR
VAR_OUTPUT
	stMotorOutput					:ST_MotorOutput;//轴的状态输出
END_VAR
VAR_INPUT
	fb_motionModule					:MotionModule;
END_VAR


Obj_Instance();
//先传递速度限制值
fb_motionModule.HMIItf.manSoftLimitVel:=fSoftLimitVel;
//
stMotorOutput.axisActualPos:=fb_motionModule.axisActualPos;
stMotorOutput.axisActualVel:=fb_motionModule.axisActualVel;
stMotorOutput.axisActualtorque:=fb_motionModule.axisActualtorque;
stMotorOutput.axisPause:=fb_motionModule.axisPause;
stMotorOutput.axisBusy:=fb_motionModule.axisBusy;
stMotorOutput.axisDone:=fb_motionModule.axisDone;
stMotorOutput.axisError:=fb_motionModule.axisError;
stMotorOutput.axisErrId:=fb_motionModule.axisErrId;
stMotorOutput.axisErrTxt:=fb_motionModule.axisErrTxt;
stMotorOutput.axisErrWTxt:=fb_motionModule.axisErrWTxt;
stMotorOutput.axisHomeState:=fb_motionModule.axisHomeState;
stMotorOutput.pAxis:=fb_motionModule.pAxis;
stMotorOutput.jogCondition:=fb_motionModule.jogCondition;
stMotorOutput.absCondition:=fb_motionModule.absCondition;
stMotorOutput.relCondition:=fb_motionModule.relCondition;
stMotorOutput.velCondition:=fb_motionModule.velCondition;
stMotorOutput.homeCondition:=fb_motionModule.homeCondition;
stMotorOutput.setCondition:=fb_motionModule.setCondition;
stMotorOutput.pMotionModule:=ADR(fb_motionModule);

(*
---If the return value is TRUE, it can be executed, and if return value is FALSE, it is not allowed; 
---Execute ABS motion; 
*)
METHOD Act_ABS : BOOL
VAR_INPUT
	pos:LREAL;//target position
	vel:LREAL;//target velocity
END_VAR
IF fb_motionModule.absCondition THEN
	fb_motionModule.absVelocity:=vel;
	fb_motionModule.absPosition:=pos;
	fb_motionModule.absExecute:=TRUE;
	Obj_Instance();
	Act_ABS:=TRUE;
ELSE
	Act_ABS:=FALSE;
END_IF
END_METHOD

(*
---If the return value is TRUE, it can be executed, and if return value is FALSE, it is not allowed; 
---Execute ABS variable motion; 
*)
METHOD Act_ABS_Mixed : BOOL
VAR_IN_OUT
	arrPos:ARRAY [*] OF LREAL;//target position array, array max length is 50
	arrVel:ARRAY [*] OF LREAL;//target velocity array, array max length is 50
END_VAR
VAR_INPUT
	//arrPos:ARRAY [1..g_Mixed_Index] OF LREAL;//target position array, array max length is 50
	//arrVel:ARRAY [1..g_Mixed_Index] OF LREAL;//target velocity array, array max length is 50
	arrLength:UINT;//array length
END_VAR
VAR
	i_Act_ABS_Mixed:UINT;
	nPosLower_Bound:DINT;//数组下标 首位
	nPosUpper_Bound:DINT;//数组下标 末位
	nPosArr_Len:DINT;//数组长度
	nVelLower_Bound:DINT;//数组下标 首位
	nVelUpper_Bound:DINT;//数组下标 末位
	nVelArr_Len:DINT;//数组长度
END_VAR
nPosLower_Bound:=LOWER_BOUND(arrPos,1);
nPosUpper_Bound:=UPPER_BOUND(arrPos,1);
nPosArr_Len:=nPosUpper_Bound-nPosLower_Bound+1;
nVelLower_Bound:=LOWER_BOUND(arrVel,1);
nVelUpper_Bound:=UPPER_BOUND(arrVel,1);
nVelArr_Len:=nVelUpper_Bound-nVelLower_Bound+1;
IF nPosArr_Len<>nVelArr_Len 
	OR nPosArr_Len>=arrLength
	OR arrLength<=0 THEN
	Act_ABS_Mixed:=FALSE;
END_IF
IF fb_motionModule.absCondition THEN
	FOR i_Act_ABS_Mixed:=1 TO arrLength BY 1 DO
		fb_motionModule.absMixedPositionArray[i_Act_ABS_Mixed]:=arrPos[nPosLower_Bound+i_Act_ABS_Mixed-1];
		fb_motionModule.absMixedVelocityArray[i_Act_ABS_Mixed]:=arrVel[nPosLower_Bound+i_Act_ABS_Mixed-1];
	END_FOR
	fb_motionModule.absMixedArrayLength:=arrLength;
	fb_motionModule.absMixedMovement:=TRUE;
	fb_motionModule.absExecute:=TRUE;
	Obj_Instance();
	Act_ABS_Mixed:=TRUE;
ELSE
	Act_ABS_Mixed:=FALSE;
END_IF
END_METHOD

(*
---If the return value is TRUE, it can be executed, and if return value is FALSE, it is not allowed; 
---Execute HOME motion; 
*)
METHOD Act_HOME : BOOL
VAR_INPUT
END_VAR
IF fb_motionModule.homeCondition THEN
	fb_motionModule.homeExecute:=TRUE;
	Obj_Instance();
	Act_HOME:=TRUE;
ELSE
	Act_HOME:=FALSE;
END_IF
END_METHOD

(*
---If the return value is TRUE, it can be executed, and if return value is FALSE, it is not allowed; 
---Execute Modulo motion; 
*)
METHOD Act_Modulo : BOOL
VAR_INPUT
	pos:LREAL;//target position
	vel:LREAL;//target velocity
END_VAR
IF fb_motionModule.moveModuloCondition THEN
	fb_motionModule.moveModuloVelocity:=vel;
	fb_motionModule.moveModuloPosition:=pos;
	fb_motionModule.moveModuloExecute:=TRUE;
	Obj_Instance();
	Act_Modulo:=TRUE;
ELSE
	Act_Modulo:=FALSE;
END_IF
END_METHOD

(*
---If the return value is TRUE, it can be executed, and if return value is FALSE, it is not allowed; 
---Execute PAUSE; 
*)
METHOD Act_PAUSE : BOOL
VAR_INPUT
END_VAR
IF TRUE THEN
	fb_motionModule.pauseExecute:=TRUE;
	Obj_Instance();
	Act_PAUSE:=TRUE;
ELSE
	Act_PAUSE:=FALSE;
END_IF
END_METHOD

(*
---If the return value is TRUE, it can be executed, and if return value is FALSE, it is not allowed; 
---Execute REL motion; 
*)
METHOD Act_REL : BOOL
VAR_INPUT
	pos:LREAL;//target position
	vel:LREAL;//target velocity
END_VAR
IF fb_motionModule.relCondition THEN
	fb_motionModule.relVelocity:=vel;
	fb_motionModule.relDistance:=pos;
	fb_motionModule.relExecute:=TRUE;
	Obj_Instance();
	Act_REL:=TRUE;
ELSE
	Act_REL:=FALSE;
END_IF
END_METHOD

(*
---If the return value is TRUE, it can be executed, and if return value is FALSE, it is not allowed; 
---Execute RESET; 
*)
METHOD Act_RESET : BOOL
VAR_INPUT
END_VAR
IF TRUE THEN
	fb_motionModule.resetExecute:=TRUE;
	Obj_Instance();
	Act_RESET:=TRUE;
ELSE
	Act_RESET:=FALSE;
END_IF
END_METHOD

(*
---If the return value is TRUE, it can be executed, and if return value is FALSE, it is not allowed; 
---Execute SetPos motion; 
*)
METHOD Act_SETPOS : BOOL
VAR_INPUT
	pos:LREAL;//target position
END_VAR
IF fb_motionModule.setCondition THEN
	fb_motionModule.setPosPosition:=pos;
	fb_motionModule.setPosExecute:=TRUE;
	Obj_Instance();
	Act_SETPOS:=TRUE;
ELSE
	Act_SETPOS:=FALSE;
END_IF
END_METHOD

(*
---If the return value is TRUE, it can be executed, and if return value is FALSE, it is not allowed; 
---Execute STOP; 
*)
METHOD Act_STOP : BOOL
VAR_INPUT
END_VAR
IF TRUE THEN
	fb_motionModule.axisStopFlag:=TRUE;
	Obj_Instance();
	Act_STOP:=TRUE;
ELSE
	Act_STOP:=FALSE;
END_IF
END_METHOD

(*
---If the return value is TRUE, it can be executed, and if return value is FALSE, it is not allowed; 
---Execute VEL motion; 
*)
METHOD Act_VEL : BOOL
VAR_INPUT
	vel:LREAL;//target velocity
	dir:BOOL;//target direction
END_VAR
IF fb_motionModule.velCondition THEN
	fb_motionModule.velVelocity:=vel;
	fb_motionModule.velDirection:=dir;
	fb_motionModule.velExecute:=TRUE;
	Obj_Instance();
	Act_VEL:=TRUE;
ELSE
	Act_VEL:=FALSE;
END_IF
END_METHOD

(*
---If the return value is TRUE, it can be executed, and if return value is FALSE, it is not allowed; 
---Execute Vel variable motion; 
*)
METHOD Act_VEL_modifyVel : BOOL
VAR_INPUT
	vel:LREAL;//target velocity
END_VAR
IF TRUE THEN
	fb_motionModule.changeVelVel(vel);
	Obj_Instance();
	Act_VEL_modifyVel:=TRUE;
ELSE
	Act_VEL_modifyVel:=FALSE;
END_IF
END_METHOD

(*
---If the return value is TRUE, it can be executed, and if return value is FALSE, it is not allowed; 
---Execute Vel stop; 
*)
METHOD Act_VEL_Stop : BOOL
VAR_INPUT
END_VAR
IF TRUE THEN
	fb_motionModule.velExecute:=FALSE;
	Obj_Instance();
	Act_VEL_Stop:=TRUE;
ELSE
	Act_VEL_Stop:=FALSE;
END_IF
END_METHOD

(*
---Get axis ABS condition
*)
METHOD Get_AbsCondition : BOOL
VAR_INPUT
END_VAR
Get_AbsCondition:=fb_motionModule.absCondition;
END_METHOD

(*
---Get axis actual position
*)
METHOD Get_ActPos : LREAL
VAR_INPUT
END_VAR
Get_ActPos:=fb_motionModule.axisActualPos;
END_METHOD

(*
---Get axis actual velocity
*)
METHOD Get_ActVel : LREAL
VAR_INPUT
END_VAR
Get_ActVel:=fb_motionModule.axisActualVel;
END_METHOD

(*
---Get axis busy state
*)
METHOD Get_Busy : BOOL
VAR_INPUT
END_VAR
Get_Busy:=fb_motionModule.axisBusy;
END_METHOD

(*
---Get axis run done signal
*)
METHOD Get_Done : BOOL
VAR_INPUT
END_VAR
Get_Done:=fb_motionModule.axisDone;
END_METHOD

(*
---Get axis abs run done signal
*)
METHOD Get_Done_Abs : BOOL
VAR_INPUT
END_VAR
Get_Done_Abs:=fb_motionModule.axisDone and ABS(fb_motionModule.axisActualPos-fb_motionModule.absPosition)<fPosDeviation;
END_METHOD

(*
---Get axis error id
*)
METHOD Get_ErrID : UDINT
VAR_INPUT
END_VAR
Get_ErrID:=fb_motionModule.axisErrId;
END_METHOD

(*
---Get axis error state
*)
METHOD Get_Error : BOOL
VAR_INPUT
END_VAR
Get_Error:=fb_motionModule.axisError;
END_METHOD

